(* IEC 61131-3 sources: ironplc-benchmarks/compat_out (part 59) *)

returs the date of january 1st for the given year
the function works for dates from 1970 - 2099

*)
(* @END_DECLARATION := '0' *)
YEAR_BEGIN := DWORD_TO_DATE(SHR(INT_TO_DWORD(y) * 1461 - 2878169,2) * 86400);

(* revision history
hm	19. dec 2007	rev 1.0
	original version

hm	4. jan 2008		rev 1.1
	formula for step7 was incorrect during leap years

hm	7. apr. 2008	rev 1.2
	deleted unused step7 code
*)

END_FUNCTION

(* @NESTEDCOMMENTS := 'Yes' *)
(* @PATH := '\/Time&Date' *)
(* @OBJECTFLAGS := '0, 8' *)
(* @SYMFILEFLAGS := '2048' *)
FUNCTION YEAR_END : DATE
VAR_INPUT
	y : INT;
END_VAR

(*
version 1.1	24. jan. 2011
programmer 	hugo
tested by	oscat

returs the date of december 31st for the given year
the function works for dates from 1970 - 2099

*)
(* @END_DECLARATION := '0' *)
YEAR_END := DWORD_TO_DATE(SHR(INT_TO_DWORD(y) * 1461 - 2876712, 2) * 86400);

(* revision history
hm	15. jun. 2008	rev 1.0
	original version

hm	24. jan 2011	rev 1.1
	improved performance
*)

END_FUNCTION

(* @NESTEDCOMMENTS := 'Yes' *)
(* @PATH := '\/Time&Date' *)
(* @OBJECTFLAGS := '0, 8' *)
(* @SYMFILEFLAGS := '2048' *)
FUNCTION YEAR_OF_DATE : INT
VAR_INPUT
	IDATE : DATE;
END_VAR

(*
version 1.4	7. oct. 2008
programmer 	hugo
tested by		oscat

returs the year of a date
the function works for dates from 1970 - 2099

*)

(* @END_DECLARATION := '0' *)
YEAR_OF_DATE := DWORD_TO_INT((DATE_TO_DWORD(idate) + 43200) / 31557600 + 1970);

(* revision history
hm	4. aug 2006		rev 1.0
	original version

hm	1. okt 2007		rev 1.1
	corrected error in algorithm
	adjustment for S7 compatibility

hm	23.12.2007		rev 1.2
	changed code for better performance

hm	7. apr. 2008	rev 1.3
	deleted unused step7 code

hm	7. oct. 2008	rev 1.4
	renamed function (year) to year_of_date

*)
END_FUNCTION

(* @NESTEDCOMMENTS := 'Yes' *)
(* @PATH := '' *)
(* @OBJECTFLAGS := '0, 8' *)
TYPE CALENDAR :
STRUCT
	UTC : DT;					(* world time UTC *)
	LDT : DT;					(* local time *)
	LDATE : DATE;				(* local date *)
	LTOD : TOD;					(* local time of day *)
	YEAR : INT;					(* year of LDATE *)
	MONTH : INT;				(* month of LDATE *)
	DAY : INT;					(* day of LDATE *)
	WEEKDAY : INT;				(* weekday of LDATE *)
	OFFSET : INT;				(* Time Zone Offset for Local time in minutes *)
	DST_EN : BOOL;				(* daylight savings time enable *)
	DST_ON : BOOL;				(* true when daylight savings time os on *)
	NAME : STRING[5];			(* name of time zone *)
	LANGUAGE : INT;			(* location number pls see location setup *)
	LONGITUDE : REAL;			(* longitude of current location *)
	LATITUDE : REAL;			(* latitude of current location *)
	SUN_RISE : TOD;				(* sun_rise for current location *)
	SUN_SET : TOD;				(* sun_set for current location *)
	SUN_MIDDAY : TOD;			(* worldtime when sun stands at south position *)
	SUN_HEIGTH : REAL	;		(* suns heigth at midday, south position *)
	SUN_HOR : REAL;			(* sun angle horizontal 0 = north in degrees *)
	SUN_VER : REAL;			(* sun angle vertical above horizon in degrees *)
	NIGHT : BOOL;				(* true between sun_set and sun_rise *)
	HOLIDAY : BOOL;			(* true when holiday *)
	HOLY_NAME : STRING[30];	(* name of holiday *)
	WORK_WEEK : INT;			(* current work week *)
END_STRUCT
END_TYPE

(* revision history
hm	21. nov. 2008	rev 1.0
	original version

hm	8. feb. 2009	rev 1.1
	added sun position data

hm	10. mar. 2009	rev 1.2
	added work_week, sun_midday, sun_heigth

hm	23. jan 2010	rev 1.3
	sun_rise, sun_set and sun_midday are now calculated in local time

*)
(* @END_DECLARATION := '0' *)

(* @NESTEDCOMMENTS := 'Yes' *)
(* @PATH := '' *)
(* @OBJECTFLAGS := '0, 8' *)
TYPE COMPLEX :
STRUCT
	re : REAL;
	im : REAL;
END_STRUCT
END_TYPE

(* revision history
hm	18. oct. 2008
	original version

*)
(* @END_DECLARATION := '0' *)

(* @NESTEDCOMMENTS := 'Yes' *)
(* @PATH := '' *)
(* @OBJECTFLAGS := '0, 8' *)
TYPE CONSTANTS_LANGUAGE :
STRUCT
	(* Language Setup *)
	DEFAULT : INT := 1; (* 1=english, 2=german 3=french *)
	LMAX : INT := 3;
	WEEKDAYS : ARRAY[1..3, 1..7] OF STRING[10] :=	['Monday', 'Tuesday', 'Wednesday', 'Thursday', 'Friday', 'Saturday', 'Sunday',
													'Montag', 'Dienstag', 'Mittwoch', 'Donnerstag', 'Freitag', 'Samstag', 'Sonntag',
													'Lundi', 'Mardi', 'Mercredi', 'Jeudi', 'Vendredi', 'Samedi', 'Dimanche'];
	WEEKDAYS2 : ARRAY[1..3, 1..7] OF STRING[2] :=	['Mo', 'Tu', 'We', 'Th', 'Fr', 'Sa', 'Su',
													'Mo', 'Di', 'Mi', 'Do', 'Fr', 'Sa', 'So',
													'Lu', 'Ma', 'Me', 'Je', 'Ve', 'Sa', 'Di'];
	MONTHS : ARRAY[1..3, 1..12] OF STRING[10] :=	['January', 'February', 'March', 'April', 'May', 'June', 'July', 'August', 'September', 'October', 'November', 'December',
													'Januar', 'Februar', 'M�rz', 'April', 'Mai', 'Juni', 'Juli', 'August', 'September', 'Oktober', 'November', 'Dezember',
													'Janvier', 'F�vrier', 'mars', 'Avril', 'Mai', 'Juin', 'Juillet', 'Ao�t', 'Septembre', 'Octobre', 'Novembre', 'Decembre'];
	MONTHS3 : ARRAY[1..3, 1..12] OF STRING[3] :=	['Jan', 'Feb', 'Mar', 'Apr', 'May', 'Jun', 'Jul', 'Aug', 'Sep', 'Oct', 'Nov', 'Dec',
													'Jan', 'Feb', 'Mrz', 'Apr', 'Mai', 'Jun', 'Jul', 'Aug', 'Sep', 'Okt', 'Nov', 'Dez',
													'Jan', 'Fev', 'Mar', 'Avr', 'Mai', 'Jun', 'Jul', 'Aou', 'Sep', 'Oct', 'Nov', 'Dec'];
	DIRS : ARRAY[1..3,0..15] OF STRING[3] :=		['N', 'NNE', 'NE', 'ENE', 'E', 'ESE', 'SE', 'SSE', 'S', 'SSW', 'SW', 'WSW', 'W', 'WNW', 'NW', 'NNW',
													'N', 'NNO', 'NO', 'ONO', 'O', 'OSO', 'SO', 'SSO', 'S', 'SSW', 'SW', 'WSW', 'W', 'WNW', 'NW', 'NNW',
													'N', 'NNO', 'NO', 'ONO', 'O', 'OSO', 'SO', 'SSO', 'S', 'SSW', 'SW', 'WSW', 'W', 'WNW', 'NW', 'NNW'];
END_STRUCT
END_TYPE

(* revision history
hm	19. oct. 2008	rev 1.0
	original version

hm	22. oct. 2008	rev 1.1
	added directions DIRS

hm	23. dec. 2008	rev 1.2
	added french language

*)
(* @END_DECLARATION := '0' *)

(* @NESTEDCOMMENTS := 'Yes' *)
(* @PATH := '' *)
(* @OBJECTFLAGS := '0, 8' *)
TYPE CONSTANTS_LOCATION :
STRUCT
	(* location setup *)
	DEFAULT : INT := 1; (* 1=germany, 2=austria 3=france 4=belgium-german 5= italien-S�dtirol *)
	LMAX : INT := 5;

	(* language spoken in the location *)
	LANGUAGE : ARRAY[1..5] OF INT := [2, 2, 3, 2, 2];

END_STRUCT
END_TYPE

(* revision history
hm	20. oct. 2008	rev 1.0
	original version

hm	23. dec. 2008	rev 1.1
	added french holidays

hm	18. jan 2011	rev 1.2
	added spoken language
	deleted holidays from structure for more flexibility

*)
(* @END_DECLARATION := '0' *)

(* @NESTEDCOMMENTS := 'Yes' *)
(* @PATH := '' *)
(* @OBJECTFLAGS := '0, 8' *)
TYPE CONSTANTS_MATH :
STRUCT
	PI : REAL := 	3.14159265358979323846264338327950288;		(* Kreiszahl PI *)
	PI2 : REAL := 	6.28318530717958647692528676655900576;	(* PI * 2 *)
	PI4 : REAL :=  12.56637061435917295385057353311801152;	(* PI * 4 *)
	PI05 : REAL :=  1.5707963267949;							(* PI / 2 *)
	PI025 : REAL := 0.785398163397448;							(* PI / 4 *)
	PI_INV : REAL := 0.318309886183791;						(* 1 / PI *)
	E : REAL := 	2.71828182845904523536028747135266249;		(* Euler constant e *)
	E_INV : REAL := 0.367879441171442;							(* 1 / e *)
	SQ2 : REAL :=	1.4142135623731;							(* Wurzel von 2 *)
	FACTS : ARRAY[0..12] OF DINT := [1,1,2,6,24,120,720,5040,40320,362880,3628800,39916800,479001600];
END_STRUCT
END_TYPE

(* revision history
hm	26.10.2008	rev 1.0
	original version

hm	26. mar. 2011	rev 1.1
	added array facts
*)
(* @END_DECLARATION := '0' *)

(* @NESTEDCOMMENTS := 'Yes' *)
(* @PATH := '' *)
(* @OBJECTFLAGS := '0, 8' *)
TYPE CONSTANTS_PHYS :
STRUCT
	C : REAL := 299792458.0;				(* Lichtgeschwindigkeit in m/s *)
	E : REAL := 1.60217653E-19;				(* elementarladung in Colomb = A * s *)
	G : REAL := 9.80665; 						(* Erdbeschleunigung in m / s� *)
	T0 : REAL := -273.15;						(* absoluter Nullpunkt in �C *)
	RU : REAL := 8.314472; 					(* Universelle Gaskonstante in J / (mol � K) *)
	PN : REAL := 101325.0;					(* NormalDruck in Pa *)
END_STRUCT
END_TYPE

(* revision history
hm	18.10.2008	rev 1.0
	original version

hm	13. mar. 2009	rev 1.1
	real constants updated to new systax using dot

*)
(* @END_DECLARATION := '0' *)

(* @NESTEDCOMMENTS := 'Yes' *)
(* @PATH := '' *)
(* @OBJECTFLAGS := '0, 8' *)
TYPE CONSTANTS_SETUP :
STRUCT
	(* setup Parameters *)
	EXTENDED_ASCII : BOOL := TRUE;
	CHARNAMES : ARRAY[1..4] OF STRING[253] := [';"&quot;&&amp;<&lt;>&gt;�&euro;�&nbsp;�&iexcl;�&cent;�&pound;�&curren;�&yen;�&brvbar;�&sect;�&uml;�&copy;�&ordf;�&laquo;�&not;�&shy;�&reg;�&macr;�&deg;�&plusmn;�&sup2;�&sup3;�&acute;�&micro;�&para;�&middot;�&cedil;�&sup1;�&ordm;�&raquo;�&frac14;�&Ucirc;',
		';�&frac34;�&iquest;�&Agrave;�&Aacute;�&Acirc;�&Atilde;�&Auml;�&Aring;�&AElig;�&Ccedil;�&Egrave;�&Eacute;�&Ecirc;�&Euml;�&Igrave;�&Iacute;�&Icirc;�&Iuml;�&ETH;�&Ntilde;�&Ograve;�&Oacute;�&Ocirc;�&Otilde;�&Ouml;�&times;�&Oslash;�&Ugrave;�&Uacute;�&frac12;',
		';�&Uuml;�&Yacute;�&THORN;�&szlig;�&agrave;�&aacute;�&acirc;�&atilde;�&auml;�&aring;�&aelig;�&ccedil;�&egrave;�&eacute;�&ecirc;�&euml;�&igrave;�&iacute;�&icirc;�&iuml;�&eth;�&ntilde;�&ograve;�&oacute;�&ocirc;�&otilde;�&ouml;�&divide;�&oslash;�&ugrave;',
		';�&uacute;�&ucirc;�&uuml;�&yacute;�&thorn;�&yuml;'];
	MTH_OFS : ARRAY[1..12] OF INT := [0,31,59,90,120,151,181,212,243,273,304,334];
	DECADES : ARRAY[0..8] OF REAL := [1.0,10.0,100.0,1000.0,10000.0,10000.0,100000.0,1000000.0,10000000.0];
END_STRUCT
END_TYPE

(* revision history
hm	24.10.2008	rev 1.0
	original version

*)
(* @END_DECLARATION := '0' *)

(* @NESTEDCOMMENTS := 'Yes' *)
(* @PATH := '' *)
(* @OBJECTFLAGS := '0, 8' *)
TYPE ESR_DATA :
STRUCT
	TYP : BYTE;
	ADRESS : STRING[10];
	DS : DT;
	TS : TIME;
	DATA : ARRAY[0..7] OF BYTE;
END_STRUCT
END_TYPE

(* revision history
hm	18. oct. 2008
	original version

*)
(* @END_DECLARATION := '0' *)

(* @NESTEDCOMMENTS := 'Yes' *)
(* @PATH := '' *)
(* @OBJECTFLAGS := '0, 8' *)
TYPE FRACTION :
STRUCT
	NUMERATOR : INT;
	DENOMINATOR : INT;
END_STRUCT
END_TYPE
(* @END_DECLARATION := '0' *)

(* @NESTEDCOMMENTS := 'Yes' *)
(* @PATH := '' *)
(* @OBJECTFLAGS := '0, 8' *)
TYPE HOLIDAY_DATA :
STRUCT
	NAME : STRING[30];
	DAY : SINT;
	MONTH : SINT;
	USE : SINT;
END_STRUCT
END_TYPE

(* revision history
hm	18. oct. 2008
	original version

*)

(*	if month = 0 then F_day is the offset in days from easter
	used :0 = NOT used, 1 = used, -1..-7 menas the weekday before the specified DATE example -3 means wednesday before 23.11
*)

(* samples for Holiday data

	HOLIDAY_DE : ARRAY[0..29] OF HOLIDAY_DATA := (name := 'Neujahr', day := 1, month := 1, use := 1),
		(name := 'Heilig Drei K�nige', day := 6, month := 1, use := 1),
		(name := 'Karfreitag', day := -2, month := 0, use := 1),
		(name := 'Ostersonntag', day := 0, month := 0, use := 1),
		(name := 'Ostermontag', day := 1, month := 0, use := 1),
		(name := 'Tag der Arbeit', day := 1, month := 5, use := 1),
		(name := 'Christi Himmelfahrt', day := 39, month := 0, use := 1),
		(name := 'Pfingstsonntag', day := 49, month := 0, use := 1),
		(name := 'Pfingstmontag', day := 50, month := 0, use := 1),
		(name := 'Fronleichnam', day := 60, month := 0, use := 1),
		(name := 'Augsburger Friedensfest', day := 8, month := 8, use := 0),
		(name := 'Maria Himmelfahrt', day := 15, month := 8, use := 1),
		(name := 'Tag der Deutschen Einheit', day := 3, month := 10, use := 1),
		(name := 'Reformationstag', day := 31, month := 10, use := 0),
		(name := 'Allerheiligen', day := 1, month := 11, use := 1),
		(name := 'Buss und Bettag', day := 23, month := 11, use := 0),
		(name := '1. Weihnachtstag', day := 25, month := 12, use := 1),
		(name := '2. Weihnachtstag', day := 26, month := 12, use := 1);

	HOLIDAY_AT : ARRAY[0..29] OF HOLIDAY_DATA := (name := 'Neujahr', day := 1, month := 1, use := 1),
		(name := 'Heilig Drei K�nige', day := 6, month := 1, use := 1),
		(name := 'Karfreitag', day := -2, month := 0, use := 1),
		(name := 'Ostersonntag', day := 0, month := 0, use := 1),
		(name := 'Ostermontag', day := 1, month := 0, use := 1),
		(name := '', day := 1, month := 5, use := 0),
		(name := 'Christi Himmelfahrt', day := 39, month := 0, use := 1),
		(name := 'Pfingstsonntag', day := 49, month := 0, use := 1),
		(name := 'Pfingstmontag', day := 50, month := 0, use := 1),
		(name := 'Fronleichnam', day := 60, month := 0, use := 1),
		(name := '', day := 8, month := 8, use := 0),
		(name := 'Maria Himmelfahrt', day := 15, month := 8, use := 1),
		(name := '', day := 3, month := 10, use := 0),
		(name := '', day := 31, month := 10, use := 0),
		(name := 'Allerheiligen', day := 1, month := 11, use := 1),
		(name := 'Maria Empf�ngnis', day := 8, month := 12, use := 1),
		(name := '1. Weihnachtstag', day := 25, month := 12, use := 1),
		(name := '2. Weihnachtstag', day := 26, month := 12, use := 1);

	HOLIDAY_FR : ARRAY[0..29] OF HOLIDAY_DATA := (name := 'Nouvel an', day := 1, month := 1, use := 1),
		(name := 'St Valentin', day := 14, month := 2, use := 0),
		(name := 'Vendredi Saint (alsace)', day := -2, month := 0, use := 0),
		(name := 'Dimanche de p�ques', day := 0, month := 0, use := 1),
		(name := 'Lundi de p�ques', day := 1, month := 0, use := 1),
		(name := 'Jeudi de Ascension', day := 39, month := 0, use := 1),
		(name := 'dimanche de Pentec�te ', day := 49, month := 0, use := 1),
		(name := 'jeudi de la Trinit�', day := 60, month := 0, use := 0),
		(name := 'F�te du travail', day := 1, month := 5, use := 1),
		(name := 'Victoire 1945 ', day := 8, month := 5, use := 1),
		(name := 'Prise de La bastille', day := 14, month := 7, use := 1),
		(name := '15 Ao�t 1944', day := 15, month := 8, use := 1),
		(name := 'Halloween', day := 31, month := 10, use := 0),
		(name := 'Armistice 1918', day := 11, month := 11, use := 1),
		(name := 'No�l', day := 25, month := 12, use := 1),
		(name := 'Saint �tienne (alsace)', day := 26, month := 12, use := 0),
		(name := 'F�te de la musique', day := 21, month := 6, use := 0);

	HOLIDAY_BED : ARRAY[0..29] OF HOLIDAY_DATA :=	(name := 'Neujahr', day := 1, month := 1, use := 1),
		(name := 'Ostersonntag', day := 0, month := 0, use := 1),
		(name := 'Ostermontag', day := 1, month := 0, use := 1),
		(name := 'Tag der Arbeit', day := 1, month := 5, use := 1),
		(name := 'Christi Himmelfahrt', day := 39, month := 0, use := 1),
		(name := 'Pfingsten', day := 49, month := 0, use := 1),
		(name := 'Pfingstmontag', day := 50, month := 0, use := 1),
		(name := 'Nationalfeiertag', day := 21, month := 7, use := 1),
		(name := 'Mari� Himmelfahrt', day := 15, month := 8, use := 1),
		(name := 'Allerheiligen', day := 1, month := 11, use := 1),
		(name := 'Feiertag DG', day := 15, month := 11, use := 1),
		(name := 'Heiligabend', day := 24, month := 12, use := 1),
		(name := '1. Weihnachtstag', day := 25, month := 12, use := 1),
		(name := '2. Weihnachtstag', day := 26, month := 12, use := 1),
		(name := 'Silvester', day := 31, month := 12, use := 1);

	HOLIDAY_ITD : ARRAY[0..29] OF HOLIDAY_DATA := (name := 'Neujahr', day := 1, month := 1, use := 1),
		(name := 'Heilig Drei K�nige', day := 6, month := 1, use := 1),
		(name := 'Ostersonntag', day := 0, month := 0, use := 1),
		(name := 'Ostermontag', day := 1, month := 0, use := 1),
		(name := 'Tag der Befeiung Italiens', day := 25, month := 4, use := 1),
		(name := 'Tag der Arbeit', day := 1, month := 5, use := 1),
		(name := 'Pfingsten', day := 49, month := 0, use := 1),
		(name := 'Pfingstmontag', day := 50, month := 0, use := 1),
		(name := 'Tag der Republik Italien', day := 2, month := 6, use := 1),
		(name := 'Mari� Himmelfahrt', day := 15, month := 8, use := 1),
		(name := 'Allerheiligen', day := 1, month := 11, use := 1),
		(name := 'Mari� Empf�ngnis', day := 8, month := 12, use := 1),
		(name := 'Heiligabend', day := 24, month := 12, use := 0),
		(name := '1. Weihnachtstag', day := 25, month := 12, use := 1),
		(name := '2. Stephanstag', day := 26, month := 12, use := 1);

*)
(* @END_DECLARATION := '0' *)

(* @NESTEDCOMMENTS := 'Yes' *)
(* @PATH := '' *)
(* @OBJECTFLAGS := '0, 8' *)
TYPE REAL2 :
STRUCT
	R1 : REAL;	(* small value *)
	RX : REAL;	(* big value *)
END_STRUCT
END_TYPE

(* revision history
hm	18. oct. 2008
	original version

*)
(* @END_DECLARATION := '0' *)

(* @NESTEDCOMMENTS := 'Yes' *)
(* @PATH := '' *)
(* @OBJECTFLAGS := '0, 8' *)
TYPE SDT :
STRUCT
	YEAR : INT;
	MONTH : INT;
	DAY : INT;
	WEEKDAY : INT;
	HOUR : INT;
	MINUTE : INT;
	SECOND : INT;
	MS : INT;
END_STRUCT
END_TYPE

(* revision history
hm	18. oct. 2008
	original version

*)
(* @END_DECLARATION := '0' *)

(* @NESTEDCOMMENTS := 'Yes' *)
(* @PATH := '' *)
(* @OBJECTFLAGS := '0, 8' *)
TYPE TIMER_EVENT :
STRUCT
	TYP : BYTE;
	CHANNEL : BYTE;
	DAY : BYTE;
	START : TOD;
	DURATION : TIME;
	LAND : BYTE;
	LOR : BYTE;
	LAST : DT;
END_STRUCT
END_TYPE

(* revision history
hm	18. oct. 2008	rev 1.0
	original version

hm	26. jan. 2011	rev 1.1
	changed type of last to be DT
*)
(* @END_DECLARATION := '0' *)

(* @NESTEDCOMMENTS := 'Yes' *)
(* @PATH := '' *)
(* @OBJECTFLAGS := '0, 8' *)
TYPE VECTOR_3 :
STRUCT
	X : REAL;
	Y : REAL;
	Z : REAL;
END_STRUCT
END_TYPE

(* revision history
hm	18. oct. 2008
	original version

*)
(* @END_DECLARATION := '0' *)

(* @NESTEDCOMMENTS := 'Yes' *)
(* @GLOBAL_VARIABLE_LIST := 'Constants' *)
(* @PATH := '' *)
(* @OBJECTFLAGS := '0, 8' *)
(* @SYMFILEFLAGS := '4096' *)
VAR_GLOBAL CONSTANT
	STRING_LENGTH : INT := 250;
	LIST_LENGTH : INT := 250;
END_VAR

(* revisionhistory
hm 3. mar. 2007
	extended accuracy of pi2
	renamed T0 to Tk for better compatibility with other libraries
	renamed C t0 c0 for better compatibility

hm	2. may. 2007
	added RU universal gas constant

hm	1. oct. 2007
	added setup parameter STEP7

hm 31. oct. 2007
	added PN

hm	6. mar. 2008
	added setup Parameter EXTENDED_ASCII

hm	28. Mar. 2008
	added setup parameter STRING_LENGTH

hm	7. apr. 2008
	Deleted unused setup parameter Step7

hm	19. apr. 2008
	added setup parameter NETWORK_BUFFER_SIZE

hm	27. apr. 2008
	added PI05 and PI025

hm	18. may. 2008
	added charname lists
	renamed E to E1

hm	30. jun. 2008
	reduced size of string constants to 253 to avoid problems with target aixia DCUF

hm	21. sep. 2008
	added section language setup
	added section location setup

hm	20. oct. 2008
	changed to structured constants

hm	16. nov. 2008
	moved structured constants to global vars for compatibility reasons

hm	13. nov. 2009
	added network_buffer_short_size
	renamed network_buffer_long_size
	changed string length to 250

hm	20. jan. 2011
	removed network buffers
	added list_length
*)
(* @OBJECT_END := 'Constants' *)
(* @CONNECTIONS := Constants
FILENAME : ''
FILETIME : 0
EXPORT : 0
NUMOFCONNECTIONS : 0
*)

(* @NESTEDCOMMENTS := 'Yes' *)
(* @GLOBAL_VARIABLE_LIST := 'Globale_Variablen' *)
(* @PATH := '' *)
(* @OBJECTFLAGS := '0, 8' *)
(* @SYMFILEFLAGS := '4096' *)
VAR_GLOBAL
	MATH : CONSTANTS_MATH;
	PHYS : CONSTANTS_PHYS;
	LANGUAGE : CONSTANTS_LANGUAGE;
	SETUP : CONSTANTS_SETUP;
	LOCATION : CONSTANTS_LOCATION;
END_VAR
(* @OBJECT_END := 'Globale_Variablen' *)
(* @CONNECTIONS := Globale_Variablen
FILENAME : ''
FILETIME : 0
EXPORT : 0
NUMOFCONNECTIONS : 0
*)

(* @NESTEDCOMMENTS := 'Yes' *)
(* @GLOBAL_VARIABLE_LIST := 'Setup_Data' *)
(* @PATH := '' *)
(* @OBJECTFLAGS := '0, 8' *)
(* @SYMFILEFLAGS := '4096' *)
VAR_GLOBAL RETAIN

END_VAR

(* @OBJECT_END := 'Setup_Data' *)
(* @CONNECTIONS := Setup_Data
FILENAME : ''
FILETIME : 0
EXPORT : 0
NUMOFCONNECTIONS : 0
*)

/* LIBRARY */
/* Standard.lib 4.10.05 11:14:46 */
/* (* @LIBRARYSYMFILEINFO := '0' *) */
/* NumOfPOUs: 21 */
/* CONCAT: 0 */
/* CTD: 0 */
/* CTU: 0 */
/* CTUD: 0 */
/* DELETE: 0 */
/* F_TRIG: 0 */
/* FIND: 0 */
/* INSERT: 0 */
/* LEFT: 0 */
/* LEN: 0 */
/* MID: 0 */
/* R_TRIG: 0 */
/* REPLACE: 0 */
/* RIGHT: 0 */
/* RS: 0 */
/* RTC: 0 */
/* SEMA: 0 */
/* SR: 0 */
/* TOF: 0 */
/* TON: 0 */
/* TP: 0 */
/* NumOfGVLs: 0 */
/* END_LIBRARY */

PROGRAM test_BAND_B
VAR
    result : BYTE;
END_VAR
    result := BAND_B(X := BYTE#16#AA, B := BYTE#16#AA);
END_PROGRAM

(* ---- test_BCDC_TO_INT.st ---- *)
(* IronPLC Compatibility Library

   Provides CODESYS-specific functions that are not part of IEC 61131-3
   and not built into IronPLC, but are needed by the OSCAT library.

   These are prepended to the compilation unit when running the
   compatibility test with --lib.
*)

(* Byte_of_Dword: Extract a byte from a DWORD by index.
   N=0 is the least significant byte, N=3 is the most significant.
   CODESYS built-in, used 16 times in OSCAT. *)
FUNCTION Byte_of_Dword : BYTE
VAR_INPUT
    in : DWORD;
    N : BYTE;
END_VAR
    Byte_of_Dword := DWORD_TO_BYTE(SHR(in, BYTE_TO_INT(N) * 8));
END_FUNCTION

(* DAY_OF_WEEK: Return day of week for a DATE value.
   Returns 0=Sunday, 1=Monday, ..., 6=Saturday.
   CODESYS extension, used 12 times in OSCAT.
   DATE is seconds since 1970-01-01. Jan 1 1970 was Thursday (=4). *)
FUNCTION DAY_OF_WEEK : SINT
VAR_INPUT
    in : DATE;
END_VAR
VAR
    days : DINT;
END_VAR
    days := DWORD_TO_DINT(DATE_TO_DWORD(in) / 86400);
    DAY_OF_WEEK := DINT_TO_SINT(((days MOD 7) + 4) MOD 7);
END_FUNCTION

(* TIME: Return current PLC uptime.
   CODESYS built-in, used 2 times in OSCAT.
   NOTE: Returns T#0s stub because __SYSTEM_UP_TIME is not accessible
   from FUNCTION context. Runtime value will not be correct until
   global variable access from functions is supported. *)
FUNCTION TIME : TIME
    TIME := T#0s;
END_FUNCTION

(* @NESTEDCOMMENTS := 'Yes' *)
(* @PATH := '\/Buffer Management' *)
(* @OBJECTFLAGS := '0, 8' *)
(* @SYMFILEFLAGS := '2048' *)
FUNCTION _BUFFER_CLEAR : BOOL
VAR_INPUT
	PT : REF_TO BYTE;
	SIZE : UINT;
END_VAR
VAR
	ptw : REF_TO DWORD;
	temp: LWORD;
	end, end32 : DWORD;
END_VAR

(*
version 1.2	31. oct. 2008
programmer 	hugo
tested by	oscat

this function will initialize a given array of byte with 0.
the function needs to be called:	_buffer_clear(adr("array"),sizeof("array"));
this function will manipulate a given array.
the function manipulates the original array, it rerturnes true when finished.
because this function works with pointers its very time efficient and it needs no extra memory.

*)
(* @END_DECLARATION := '0' *)
(* this routine uses 32 bit access to gain speed *)
(* first access bytes till pointer is aligned for 32 bit access *)
temp := pt;
end := temp + UINT_TO_DWORD(size);
end32 := end - 3;
WHILE (pt < end) AND ((temp AND 16#00000003) > 0) DO
	pt^ := 0;
	pt := pt + 1;
	temp := temp + 1;
END_WHILE;
(* pointer is aligned, now copy 32 bits at a time *)
ptw := pt;
WHILE ptw < end32 DO (* *)
	ptw^ := 0;
	ptw := ptw + 4;
END_WHILE;
(* copy the remaining bytes in byte mode *)
pt := ptw;
WHILE pt < end DO
	pt^ := 0;
	pt := pt + 1;
END_WHILE;

_BUFFER_CLEAR := TRUE;

(* revision History
hm 	5. mar. 2008	rev 1.0
	original version

hm	16. mar. 2008	rev 1.1
	added type conversion to avoid warnings under codesys 30
	chaged type of input size to uint
	deleted unused variable i

hm	31. oct. 2008	rev 1.2
	corrected an error while routine would write outside of arrays

*)
END_FUNCTION

(* @NESTEDCOMMENTS := 'Yes' *)
(* @PATH := '\/Buffer Management' *)
(* @OBJECTFLAGS := '0, 8' *)
(* @SYMFILEFLAGS := '2048' *)
FUNCTION _BUFFER_INIT : BOOL
VAR_INPUT
	PT : REF_TO BYTE;
	SIZE : UINT;
	INIT : BYTE;
END_VAR
VAR
	ptw : REF_TO DWORD;
	temp : LWORD;
	end, end32 : DWORD;
END_VAR

(*
version 1.2	31. oct. 2008
programmer 	hugo
tested by	oscat

this function will initialize a given array of byte with init.
the function needs to be called:	_buffer_init(adr("array"),sizeof("array"),init);
this function will manipulate a given array.
the function manipulates the original array, it rerturnes true when finished.
because this function works with pointers its very time efficient and it needs no extra memory.

*)
(* @END_DECLARATION := '0' *)
(* this routine uses 32 bit access to gain speed *)
(* first access bytes till pointer is aligned for 32 bit access *)
temp := pt;
end := temp + UINT_TO_DWORD(size);
end32 := end - 3;
WHILE (pt < end) AND ((temp AND 16#00000003) > 0) DO
	pt^ := init;
	pt := pt + 1;
	temp := temp + 1;
END_WHILE;
(* pointer is aligned, now copy 32 bits at a time *)
ptw := pt;
temp := SHL(BYTE_TO_DWORD(init),24) OR SHL(BYTE_TO_DWORD(init),16) OR SHL(BYTE_TO_DWORD(init),8) OR BYTE_TO_DWORD(init);
WHILE ptw < end32 DO
	ptw^ := temp;
	ptw := ptw + 4;
END_WHILE;
(* copy the remaining bytes in byte mode *)
pt := ptw;
WHILE pt < end DO
	pt^ := init;
	pt := pt + 1;
END_WHILE;

_BUFFER_INIT := TRUE;

(* revision History
hm 	5. mar. 2008	rev 1.0
	original version

hm	16. mar. 2008	rev 1.1
	added type conversion to avoid warnings under codesys 3.0
	chaged type of input size to uint.

hm	31. oct. 2008	rev 1.2
	corrected an error while routine would write outside of arrays

*)
END_FUNCTION

(* @NESTEDCOMMENTS := 'Yes' *)
(* @PATH := '\/Buffer Management' *)
(* @OBJECTFLAGS := '0, 8' *)
(* @SYMFILEFLAGS := '2048' *)
FUNCTION _BUFFER_INSERT : INT
VAR_INPUT
	STR : STRING[STRING_LENGTH];
	POS : INT;
	PT : REF_TO ARRAY[0..32767] OF BYTE;
	SIZE : UINT;
END_VAR
VAR
	end : INT;
	lx: INT;
	i: INT;
END_VAR

(*
version 1.5	2. jan. 2012
programmer 	hugo
tested by	oscat

this function will insert a string at a given position in a buffer.
the function needs to be called:	_buffer_init(adr("array"),sizeof("array"),init);
this function will manipulate a given array.
the function manipulates the original array, it returnes the next position after the input string when finished.
because this function works with pointers its very time efficient and it needs no extra memory.

*)
(* @END_DECLARATION := '0' *)
lx := LEN(str);
end := pos + lx;
(* first move the upper part of the buffer to make space for the string *)
FOR i := UINT_TO_INT(size) - 1 TO end BY -1 DO
	pt^[i] := pt^[i-lx];
END_FOR;
(* copy the string *)
_BUFFER_INSERT := _STRING_TO_BUFFER(str, pos, PT, size);

(* revision History
hm 	9. mar. 2008	rev 1.0
	original version

hm	16. mar. 2008	rev 1.1
	changed type of input size to uint

hm	13. may. 2008	rev 1.2
	changed type of pointer to array[1..32767]
	changed size of string to STRING_LENGTH

hm	23. mar. 2009	rev 1.3
	avoid writing to input pos

hm	12. nov. 2009	rev 1.4
	code optimized

hm 2. jan 2012	rev 1.5
	function now returns the next position after the input string

*)
END_FUNCTION

(* @NESTEDCOMMENTS := 'Yes' *)
(* @PATH := '\/Buffer Management' *)
(* @OBJECTFLAGS := '0, 8' *)
(* @SYMFILEFLAGS := '2048' *)
FUNCTION _BUFFER_UPPERCASE : BOOL
VAR_INPUT
	PT : REF_TO ARRAY[0..32000] OF BYTE;
	SIZE : INT;
END_VAR
VAR
	pos: INT;
END_VAR

(*
version 1.0	20. jan. 2011
programmer 	hugo
tested by	oscat

this function will convert an array of byte into uppercase
the function needs to be called:	_buffer_clear(adr("array"),sizeof("array"));
this function will manipulate a given array.
the function manipulates the original array, it rerturnes true when finished.
because this function works with pointers its very time efficient and it needs no extra memory.

*)
(* @END_DECLARATION := '0' *)
pos := 0;
WHILE pos < size DO
	PT^[pos] := TO_UPPER(pt^[pos]);
	pos := pos + 1;
END_WHILE;

_BUFFER_UPPERCASE := TRUE;

(* revision History
hm 	20. jan. 2011	rev 1.0
	original version

*)
END_FUNCTION

(* @NESTEDCOMMENTS := 'Yes' *)
(* @PATH := '\/Buffer Management' *)
(* @OBJECTFLAGS := '0, 8' *)
(* @SYMFILEFLAGS := '2048' *)
FUNCTION _STRING_TO_BUFFER : INT
VAR_INPUT
	STR : STRING[STRING_LENGTH];
	POS : INT;
	PT : REF_TO ARRAY[0..32767] OF BYTE;
	SIZE : UINT;
END_VAR
VAR
	ps : REF_TO BYTE;
	i: INT;
	end: INT;
END_VAR

(*
version 1.4	2. jan. 2012
programmer 	hugo
tested by		oscat

this function will copy a string into an array of byte starting at position pos.
the function needs to be called:	_String_To_buffer(str, pos, adr("array"),sizeof("array"));
this function will manipulate the array directly in memory and returns the position after the input string when finished.
because this function works with pointers its very time efficient and it needs no extra memory.

*)
(* @END_DECLARATION := '0' *)
ps := REF(str);
end := MIN(pos + LEN(str), UINT_TO_INT(size));
IF end > 0 THEN end := end -1; END_IF;
FOR i := pos TO end DO
	pt^[i] := ps^;
	ps := ps + 1;
END_FOR;

_STRING_TO_BUFFER := i;

(* revision History

hm 	5. mar. 2008	rev 1.0
	original version

hm	16. mar. 2008	rev 1.1
	changed type of input size to uint

hm	13. may. 2008	rev 1.2
	changed type of pointer to array[1..32767]
	changed size of string to STRING_LENGTH

hm	12. nov. 2009	rev 1.3
	limit end to size - 1

hm	2. jan 2012	rev 1.4
	return the position after the input string when finished
*)
END_FUNCTION

(* @NESTEDCOMMENTS := 'Yes' *)
(* @PATH := '\/Buffer Management' *)
(* @OBJECTFLAGS := '0, 8' *)
(* @SYMFILEFLAGS := '2048' *)
FUNCTION BUFFER_COMP : INT
VAR_INPUT
	PT1 : REF_TO ARRAY[0..32767] OF BYTE;
	SIZE1 : INT;
	PT2 : REF_TO ARRAY[0..32767] OF BYTE;
	SIZE2 : INT;
	START : INT;
END_VAR
VAR
	i, j, end : INT;
	firstbyte: BYTE;
END_VAR

(*
version 1.1	12. nov. 2009
programmer 	hugo
tested by	oscat

*)
(* @END_DECLARATION := '0' *)
(* search for first character match *)
IF size2 <= size1 THEN
	end := size1 - size2;
	firstbyte := PT2^[0];
	FOR i := START TO end DO
		IF PT1^[i] = firstbyte THEN
			(* first character matches, now compare rest of array *)
			j := 1;
			WHILE j < size2 DO
				IF pt2^[j] <> pt1^[j+i] THEN EXIT; END_IF;
				j := j + 1;
			END_WHILE;
			(* when J > size2 a match was found return the position i in buffer1 *)
			IF j = size2 THEN
				BUFFER_COMP := i;
				RETURN;
			END_IF;
		END_IF;
	END_FOR;
END_IF;
BUFFER_COMP := -1;

(*
hm 14. nov. 2008	rev 1.0
	original version

hm	12. nov. 2009	rev 1.1
	performance increase

*)
END_FUNCTION

(* @NESTEDCOMMENTS := 'Yes' *)
(* @PATH := '\/Buffer Management' *)
(* @OBJECTFLAGS := '0, 8' *)
(* @SYMFILEFLAGS := '2048' *)
FUNCTION BUFFER_SEARCH : INT
VAR_INPUT
	PT : REF_TO ARRAY[0..32767] OF BYTE;
	SIZE : INT;
	STR : STRING[STRING_LENGTH];
	POS : INT;
	IGN : BOOL;
END_VAR
VAR
	ps : REF_TO ARRAY[0..STRING_LENGTH] OF BYTE;
	chx : BYTE;
	i: INT;
	end: INT;
	k: INT;
	lx: INT;
END_VAR

(*
version 1.4	25. jan 2011
programmer 	hugo
tested by	oscat

this function will search for a string STR in an array of byte starting at position pos.
the function needs to be called: buffer_search(adr("array"),sizeof("array"), STR, POS, IGN);
because this function works with pointers its very time efficient and it needs no extra memory.
The function returns the position of the first character of the string in the array if found.
a -1 is returned if the string is not found in the array.
when IGN = TRUE, STR must be in capital letters and the search is case insensitv.

*)
(* @END_DECLARATION := '0' *)
ps := REF(STR);
lx := LEN(STR);
end := MIN(SIZE - lx, SIZE - 1);
lx := lx - 1;
FOR i := pos TO end DO
	FOR k := 0 TO lx DO
		IF IGN THEN chx := TO_UPPER(pt^[i+k]); ELSE chx := pt^[i+k]; END_IF;
		IF ps^[k] <> chx THEN EXIT; END_IF;
	END_FOR;
	IF k > lx THEN
		BUFFER_SEARCH := i;
		RETURN;
	END_IF;
END_FOR;
BUFFER_SEARCH := -1;

(* revision History

hm 5. mar. 2008	rev 1.0
	original version

hm	16. mar. 2008	rev 1.1
	chaged type of input size to uint

hm	13. may. 2008	rev 1.2
	changed type of pointer to array[1..32767]
	changed size of string to STRING_LENGTH

hm	12. nov. 2009	rev 1.3
	limit end to array size

hm	25. jan. 2011	rev 1.4
	ign = True will now ignore case
	return -1 if nothing found
*)
END_FUNCTION

(* @NESTEDCOMMENTS := 'Yes' *)
(* @PATH := '\/Buffer Management' *)
(* @OBJECTFLAGS := '0, 8' *)
(* @SYMFILEFLAGS := '2048' *)
FUNCTION BUFFER_TO_STRING : STRING[STRING_LENGTH]
VAR_INPUT
	PT : REF_TO ARRAY[0..32767] OF BYTE;
	SIZE : UINT;
	START : UINT;
	STOP : UINT;
END_VAR
VAR
	ps : REF_TO BYTE;
	i : UINT;
	stp: UINT;
	sta: UINT;
END_VAR

(*
version 1.5	12. nov. 2009
programmer 	hugo
tested by		oscat

this function will retrieve a string from an array of byte starting at position start and stop at position stop.
the function needs to be called:	buffer_TO_String(adr("array"),sizeof("array"), start, stop);
because this function works with pointers its very time efficient and it needs no extra memory.

*)
(* @END_DECLARATION := '0' *)
ps := REF(BUFFER_TO_STRING);
IF size = 0 THEN RETURN; END_IF;
sta := MIN(start, size -1);
stp := MIN(stop, size -1);

(* check for maximum string_length *)
IF UINT_TO_INT(stp - sta + 1) >= STRING_LENGTH THEN
	stp := sta + INT_TO_UINT(STRING_LENGTH) - 1;
END_IF;

FOR i := sta TO stp DO
	ps^ := pt^[i];
	ps := ps + 1;
END_FOR;

(* terminate the string *)

ps^ := 0;

(* revision History
hm 	5. mar. 2008	rev 1.0
	original version

hm	16. mar. 2008	rev 1.1
	changed type of input size to uint

hm	13. may. 2008	rev 1.2
	changed type of pointer to array[0..32767]
	changed size of string to STRING_LENGTH

hm	12. jun. 2008	rev 1.3
	check for pointer overrun
	change input start and stop to uint
	added type conversions to avoid warnings under codesys 3.0

hm	23. mar. 2009	rev 1.4
	avoid writing to input stop

hm	12. nov. 2009 rev 1.5
	limit start and stop to size -1

*)
END_FUNCTION

(* @NESTEDCOMMENTS := 'Yes' *)
(* @PATH := '\/Engineering\/automation' *)
(* @OBJECTFLAGS := '0, 8' *)
(* @SYMFILEFLAGS := '2048' *)
FUNCTION_BLOCK DRIVER_1
VAR_INPUT (* CONSTANT *)
	Toggle_Mode : BOOL;
	Timeout : TIME;
END_VAR
VAR_INPUT
	SET0 : BOOL;
	IN : BOOL;
	RST : BOOL;
END_VAR
VAR_OUTPUT
	Q : BOOL;
END_VAR
VAR
	off : TON;
	edge: BOOL;
END_VAR

(*
version 1.0	2 jan 2008
programmer 	hugo
tested by		tobias

driver_1 is a multi purpose driver.
a rising edge on in sets the output high if toggle is flase. while toggle is true, a rising edge on in toggles the output Q.
if a timeout is specified the output q will be reset to false automatically after the timeout has elapsed.
a asynchronous reset and set will force the output high or low respectively.

*)
(* @END_DECLARATION := '0' *)
IF off.Q THEN Q := FALSE; END_IF;
IF rst THEN
	Q := FALSE;
ELSIF set0 THEN
	Q := TRUE;
ELSIF IN AND NOT edge THEN
	IF toggle_mode THEN q := NOT Q; ELSE q := TRUE; END_IF;
END_IF;
edge := in;
IF timeout > t#0s THEN off(in := Q, PT := Timeout); END_IF;

(* revision history
hm	2. jan 2008		rev 1.0
	original version

*)
END_FUNCTION_BLOCK

(* @NESTEDCOMMENTS := 'Yes' *)
(* @PATH := '\/Engineering\/automation' *)
(* @OBJECTFLAGS := '0, 8' *)
(* @SYMFILEFLAGS := '2048' *)
FUNCTION_BLOCK DRIVER_4
VAR_INPUT (* CONSTANT *)
	Toggle_Mode : BOOL;
	Timeout : TIME;
END_VAR
VAR_INPUT
	SET0 : BOOL;
	IN0, IN1, IN2, IN3 : BOOL;
	RST : BOOL;
END_VAR
VAR_OUTPUT
	Q0, Q1, Q2, Q3 : BOOL;
END_VAR
VAR
	d0, d1, d2, d3 : DRIVER_1;
END_VAR

(*
version 1.0	2 jan 2008
programmer 	hugo
tested by		tobias

driver_4 is a 4 channel multi purpose driver.
a rising edge on in? sets the output Q? high if toggle_mode is flase. while toggle_mode is true, a rising edge on in? toggles the output Q?.
if a timeout is specified the output Q? will be reset to false automatically after the timeout has elapsed.
a asynchronous reset and set will force the output high or low respectively.
an asynchronous set will force all outputs high simultaneously

*)
(* @END_DECLARATION := '0' *)
D0(Set0:=set0, in:=in0, rst:=rst, toggle_mode:=toggle_mode, timeout:=timeout);
D1(Set0:=set0, in:=in1, rst:=rst, toggle_mode:=toggle_mode, timeout:=timeout);
D2(Set0:=set0, in:=in2, rst:=rst, toggle_mode:=toggle_mode, timeout:=timeout);
D3(Set0:=set0, in:=in3, rst:=rst, toggle_mode:=toggle_mode, timeout:=timeout);
Q0 := D0.Q;
Q1 := D1.Q;
Q2 := D2.Q;
Q3 := D3.Q;

(* revision history
hm	2. jan 2008		rev 1.0
	original version

*)
END_FUNCTION_BLOCK

(* @NESTEDCOMMENTS := 'Yes' *)
(* @PATH := '\/Engineering\/automation' *)
(* @OBJECTFLAGS := '0, 8' *)
(* @SYMFILEFLAGS := '2048' *)
FUNCTION_BLOCK DRIVER_4C
VAR_INPUT
	IN : BOOL;
	RST : BOOL;
END_VAR
VAR_INPUT (* CONSTANT *)
	Timeout : TIME;
	SX : ARRAY[1..7] OF BYTE := [1,3,7,15];
END_VAR
VAR_OUTPUT
	SN : INT;
	Q0 : BOOL;
	Q1 : BOOL;
	Q2 : BOOL;
	Q3 : BOOL;
END_VAR
VAR
	off : TON;
	edge: BOOL;
END_VAR

(*
version 1.0	23. mar. 2009
programmer 	hugo
tested by	tobias

driver_4C is a multi purpose driver.
a rising edge on in switches from S0 state S1 and the next edge to state S2 and so on.
in state S0 all outputs Q are FALSE.
The stet of the Outputs in any state S? is configurable with setup variables.
The variables S1..S5 define the states, while the sequence is terminated when a state Variable S? = 0.
The lower bits 0..3 of the state vars S? are corresponding to the Outputs Q0..Q3

*)
(* @END_DECLARATION := '0' *)
IF RST OR off.Q THEN
	SN := 0;
ELSIF IN AND NOT edge THEN
	SN := SN + 1;
	IF SN > 7 OR SX[SN] = 0 THEN SN := 0; END_IF;
END_IF;
edge := in;
IF SN > 0 THEN
	Q0 := SX[SN].0;
	Q1 := SX[SN].1;
	Q2 := SX[SN].2;
	Q3 := SX[SN].3;
ELSE
	Q0 := FALSE;
	Q1 := FALSE;
	Q2 := FALSE;
	Q3 := FALSE;
END_IF;

(* maximaum timeout *)
IF timeout > t#0s THEN off(in := SN > 0, PT := Timeout); END_IF;

(* revision history
hm	23. mar. 2009	rev 1.0
	original version

*)
END_FUNCTION_BLOCK

(* @NESTEDCOMMENTS := 'Yes' *)
(* @PATH := '\/Engineering\/automation' *)
(* @OBJECTFLAGS := '0, 8' *)
(* @SYMFILEFLAGS := '2048' *)
 FUNCTION_BLOCK FLOW_CONTROL
VAR_INPUT
	IN : BOOL;
	REQ : BOOL;
	ENQ : BOOL;
	RST : BOOL;
END_VAR
VAR_INPUT (* CONSTANT *)
	T_AUTO : TIME := T#1h;
	T_DELAY : TIME := T#23h;
END_VAR
VAR_OUTPUT
	Q : BOOL;
	STATUS : BYTE;
END_VAR
VAR
	timer : TP_1D;
END_VAR

(*
version 1.0	28. jun. 2008
programmer 	hugo
tested by	oscat

FLOW_CONTROL switches a valves depending on the input in.
flow control also limits the maximum ontime of the valve and controls pressure on the output side.

*)

(* @END_DECLARATION := '0' *)
STATUS := 100;
IF RST THEN
	Q := FALSE;
	timer(rst := TRUE);
	timer.RST := FALSE;
	STATUS := 103;
ELSIF ENQ THEN
	IF IN THEN
		status := 101;
	END_IF;
	IF REQ THEN
		(* timer will generate a timed pulse after TP goes high *)
		timer.PT1 := T_AUTO;
		timer.PTD := T_DELAY;
		timer.IN := TRUE;
		STATUS := 102;
	END_IF;
END_IF;

(* set output and run timer *)
timer();
timer.IN := FALSE;
Q := (IN AND ENQ) OR timer.Q;

(* revision history
hm 	28. jun. 2008 	rev 1.0
	original version

*)
END_FUNCTION_BLOCK

(* @NESTEDCOMMENTS := 'Yes' *)
(* @PATH := '\/Engineering\/automation' *)
(* @OBJECTFLAGS := '0, 8' *)
(* @SYMFILEFLAGS := '2048' *)
FUNCTION_BLOCK FT_Profile
VAR_INPUT
	K : REAL := 1.0;
	O : REAL;
	M : REAL := 1.0;
	E : BOOL;
END_VAR
VAR_INPUT (* CONSTANT *)
	value_0 : REAL;
	time_1 : TIME;
	value_1 : REAL;
	time_2 : TIME;
	value_2 : REAL;
	time_3 : TIME;
	value_3 : REAL;
	time_10 : TIME;
	value_10 : REAL;
	time_11 : TIME;
	value_11 : REAL;
	time_12 : TIME;
	value_12 : REAL;
	time_13 : TIME;
	value_13 : REAL;
END_VAR
VAR_OUTPUT
	Y : REAL;
	RUN : BOOL;
	ET : TIME;
END_VAR
VAR
	tx : TIME;
	edge : BOOL;
	state: BYTE;
	ta: TIME;
	tb: TIME;
	t0 : TIME;
	temp: REAL;
	va: REAL;
	vb: REAL;
END_VAR

(*
version 1.1	15 sep 2007
programmer 	tobias
tested by		hugo

FT_Profile generates an output signal which is defined by values over a time scale.
the different values are connected by ramps between the individual values.
a rising edge on E starts the output signal generation and E = True can delay time_3 / value_3 as long as it stays true.
an additional multiplier K can be used to multiply the output and an offset O can be added to the output dynamically.
*)
(* @END_DECLARATION := '0' *)
(* read system time *)
tx := DWORD_TO_TIME(T_PLC_MS());

(* determine start condition *)
IF E AND NOT edge THEN
	RUN := TRUE;
	ET := t#0s;
	t0 := tx;
	ta := tx;
	tb := multime(time_1, M);
	va := value_0;
	vb := value_1;
	temp := value_0;
	state := 1;
END_IF;
edge := E;

(* generate startup profile *)
IF run THEN
	CASE state OF
		1:	IF tx - ta >= tb THEN
				ta := ta + tb;
				tb := multime(time_2 - time_1, M);
				va := value_1;
				vb := value_2;
				temp := value_1;
				state := 2;
			ELSE
				temp := ((vb - va) * TIME_TO_REAL(tx - ta) / TIME_TO_REAL(tb) + va);
			END_IF;
		2:	IF tx - ta >= tb THEN
				ta := ta + tb;
				tb := multime(time_3 - time_2, M);
				va := value_2;
				vb := value_3;
				temp := value_2;
				state := 3;
			ELSE
				temp := ((vb - va) * TIME_TO_REAL(tx - ta) / TIME_TO_REAL(tb) + va);
			END_IF;
		3:	IF tx - ta >= tb THEN
				ta := ta + tb;
				tb := multime(time_10 - time_3, M);
				va := value_3;
				vb := value_10;
				temp := value_3;
				state := 4;
			ELSE
				temp := ((vb - va) * TIME_TO_REAL(tx - ta) / TIME_TO_REAL(tb) + va);
			END_IF;
		4 :	IF tx - ta >= tb THEN
				ta := ta + tb;
				tb := multime(time_11 - time_10, M);
				va := value_10;
				vb := value_11;
				temp := value_10;
				IF E THEN state := 5; ELSE state := 6; END_IF;
			ELSE
				temp := ((vb - va) * TIME_TO_REAL(tx - ta) / TIME_TO_REAL(tb) + va);
			END_IF;
		5:	(* extend the signal while E is true *)
			IF E THEN
				ta := tx;
			ELSE
				state := 6;
			END_IF;
		6:	IF tx - ta >= tb THEN
				ta := ta + tb;
				tb := multime(time_12 - time_11, M);
				va := value_11;
				vb := value_12;
				temp := value_11;
				state := 7;
			ELSE
				temp := ((vb - va) * TIME_TO_REAL(tx - ta) / TIME_TO_REAL(tb) + va);
			END_IF;
		7:	IF tx - ta >= tb THEN
				ta := ta + tb;
				tb := multime(time_13 - time_12, M);
				va := value_12;
				vb := value_13;
				temp := value_12;
				state := 8;
			ELSE
				temp := ((vb - va) * TIME_TO_REAL(tx - ta) / TIME_TO_REAL(tb) + va);
			END_IF;
		8:	IF tx - ta >= tb THEN
				temp := value_13;
				run := FALSE;
			ELSE
				temp := ((vb - va) * TIME_TO_REAL(tx - ta) / TIME_TO_REAL(tb) + va);
			END_IF;
	END_CASE;
	Y := temp * K + O;
	ET := tx - t0;
END_IF;

(* revision history
hm	27 feb 2007		rev 1.0
	original version

hm	15. sep2007		rev 1.1
	replaced Time() with T_PLC_MS for compatibility and performance reasons

*)
END_FUNCTION_BLOCK

(* @NESTEDCOMMENTS := 'Yes' *)
(* @PATH := '\/Engineering\/automation' *)
(* @OBJECTFLAGS := '0, 8' *)
(* @SYMFILEFLAGS := '2048' *)
FUNCTION_BLOCK INC_DEC
VAR_INPUT
	CHa : BOOL;
	CHb : BOOL;
	RST : BOOL;
END_VAR
VAR_OUTPUT
	dir : BOOL;
	cnt : INT;
END_VAR
VAR
	edgea : BOOL;
	clk: BOOL;
	clka: BOOL;
	clkb: BOOL;
	edgeb: BOOL;
	axb: BOOL;
END_VAR

(*
	version 1.0	4 aug 2006
	programmer 	oscat
	tested BY		oscat

incremental decoder with quadruple accuracy.
2 pulses for each channel are created for each directional pulse.
*)
(* @END_DECLARATION := '0' *)
axb := cha XOR chb;

(* create pulses for channel a *)
clka := cha XOR edgea;
edgea := cha;

clkb := chb XOR edgeb;
edgeb := chb;

(* create pulses for both channels *)
clk := clka OR clkb;

(* set the direction output *)
IF axb AND clka THEN dir := TRUE; END_IF;
IF axb AND clkb THEN dir := FALSE; END_IF;

(* increment or decrement the counter *)
IF clk AND dir THEN cnt := cnt + 1; END_IF;
IF clk AND NOT dir THEN cnt := cnt -1; END_IF;

(* reset the counter if rst active *)
IF rst THEN cnt := 0; END_IF;

END_FUNCTION_BLOCK

(* @NESTEDCOMMENTS := 'Yes' *)
(* @PATH := '\/Engineering\/automation' *)
(* @OBJECTFLAGS := '0, 8' *)
(* @SYMFILEFLAGS := '2048' *)
FUNCTION_BLOCK INTERLOCK
VAR_INPUT
	I1, I2 : BOOL;
	TL : TIME;
END_VAR
VAR_OUTPUT
	Q1, Q2 : BOOL;
END_VAR
VAR
	T1, T2 : TOF;
END_VAR

(*
version 1.0	28 sep 2007
programmer 	hugo
tested by		tobias

INTERLOCK has two inputs I1 and I2 which drive the corresponding outputs Q1 and Q2.
the inputs signals lock each other out and therfore I1 can only drive Q1 when I2 is Low and vice versa.
The input TL specifies a dead time between two outputs can become active.
an output can only become active when the other output was not active for the time TL.

*)
(* @END_DECLARATION := '0' *)
(* the input signal have a run delay to lockout the other input *)
T1(IN := I1, PT := TL);
T2(IN := I2, PT := TL);

Q1 := I1 AND NOT t2.Q;
Q2 := I2 AND NOT t1.Q;

(* revision history

hm	28 sep 2007		rev 1.0
	original version

*)
END_FUNCTION_BLOCK

(* @NESTEDCOMMENTS := 'Yes' *)
(* @PATH := '\/Engineering\/automation' *)
(* @OBJECTFLAGS := '0, 8' *)
(* @SYMFILEFLAGS := '2048' *)
FUNCTION_BLOCK INTERLOCK_4
VAR_INPUT (* CONSTANT *)
END_VAR
VAR_INPUT
	I0 : BOOL;
	I1 : BOOL;
	I2 : BOOL;
	I3 : BOOL;
	E : BOOL;
	MODE : INT;

END_VAR
VAR_OUTPUT
	OUT : BYTE;
	TP : BOOL;
END_VAR
VAR
	in: BYTE;
	last: BYTE;
	old: BYTE;
	lmode: INT;
END_VAR

(*
version 1.1	14. mar. 2009
programmer 	hugo
tested by		oscat

INTERLOCK_4 detects one of 4 switches and delivers the number of the switch pressed on the output out
a output tp is true for one cycle if the output has changed.
a setup variable MODE selects between 3 different modes:
MODE = 0, any input active will disable all other inputs
MODE = 1, the input with the highest number will be acepted
mode = 2, the input last pressed will disable all others

*)
(* @END_DECLARATION := '0' *)
(* check if enable is active *)
IF E THEN
(* reset all vars when there is a mode change on thy fly *)
	IF mode <> lmode THEN
		out := 0;
		last := 0;
		old := 0;
		lmode := mode;
	END_IF;
	(* load inputs into in *)
	in.0 := I0;
	in.1 := I1;
	in.2 := I2;
	in.3 := I3;
	(* only execute when there is any change *)
	IF in <> last THEN
		(* only execute when inputs have chages state *)
		CASE mode OF
			0:	(* output directly display inputs as bits in byte out *)
				out := in;

			1:	(* the input with the highest number will be acepted *)
				IF in.3 THEN out := 8;
				ELSIF in.2 THEN out := 4;
				ELSIF in.1 THEN out := 2;
				ELSE out := in;
				END_IF;

			2:	(* input last pressed will be displayed only *)
				last := ((in XOR last) AND in);
				IF last.3 THEN out := 8;
				ELSIF last.2 THEN out := 4;
				ELSIF last.1 THEN out := 2;
				ELSE out := last;
				END_IF;

			3:	(* any input active will disable all other inputs *)
				IF (out AND in) = 0 THEN
					IF in.3 THEN out := 8;
					ELSIF in.2 THEN out := 4;
					ELSIF in.1 THEN out := 2;
					ELSE out := in;
					END_IF;
				END_IF;

		END_CASE;
		last := in;
	END_IF;
	tp := out <> old;
	old := out;
ELSE
	out := 0;
	last := 0;
	old := 0;
	lmode := 0;
	tp := FALSE;
END_IF;

(* revision history
hm	24. oct 2008	rev 1.0
	original version

hm	14. mar. 2009	rev 1.1
	replaced double assignments

*)
END_FUNCTION_BLOCK

(* @NESTEDCOMMENTS := 'Yes' *)
(* @PATH := '\/Engineering\/automation' *)
(* @OBJECTFLAGS := '0, 8' *)
(* @SYMFILEFLAGS := '2048' *)
FUNCTION MANUAL : BOOL
VAR_INPUT
	IN : BOOL;
	ON : BOOL;
	OFF : BOOL;
END_VAR

(*
version 1.0	21. nov. 2008
programmer 	hugo
tested by	oscat

MANUAL is a manual override for digital signals.
when on and off = FALSE, the output follows IN.
ON = TRUE forces the output high, and OFF = TRUE forces the output low.

*)
(* @END_DECLARATION := '0' *)
MANUAL := NOT OFF AND (IN OR ON);

(* revision history
hm	21. nov 2008	rev 1.0
	original version

*)
END_FUNCTION

(* @NESTEDCOMMENTS := 'Yes' *)
(* @PATH := '\/Engineering\/automation' *)
(* @OBJECTFLAGS := '0, 8' *)
(* @SYMFILEFLAGS := '2048' *)
FUNCTION_BLOCK MANUAL_1
VAR_INPUT
	IN : BOOL;
	MAN : BOOL;
	M_I : BOOL;
	SET0 : BOOL;
	RST : BOOL;
END_VAR
VAR_OUTPUT
	Q : BOOL;
	STATUS : BYTE;
END_VAR
VAR
	S_edge : BOOL;
	r_edge : BOOL;
	edge: BOOL;
END_VAR

(*
version 1.2	14. mar. 2009
programmer 	hugo
tested by		oscat

MANUAL_1 is a manual override for digital signals.
When MAN = FALSE, the output follows IN and when MAN = TRUE the Output follows M_I.

*)
(* @END_DECLARATION := '0' *)
IF NOT man THEN
	Q := IN;
	STATUS := 100;
	edge := FALSE;
ELSIF NOT s_edge AND set0 THEN
	Q := TRUE;
	edge := TRUE;
	status := 101;
ELSIF NOT r_edge AND rst THEN
	Q := FALSE;
	edge := TRUE;
	status := 102;
ELSIF NOT edge THEN
	Q := M_I;
	status := 103;
END_IF;

(* remember levels of manual signals *)
s_edge := SET0;
r_edge := RST;

(* revision history
hm	17. jun 2008	rev 1.0
	original version

hm	17. oct 2008	rev 1.1
	deleted unnecessary variable m_edge

hm	14. mar. 2009	rev 1.2
	replaced double assignments

*)
END_FUNCTION_BLOCK

(* @NESTEDCOMMENTS := 'Yes' *)
(* @PATH := '\/Engineering\/automation' *)
(* @OBJECTFLAGS := '0, 8' *)
(* @SYMFILEFLAGS := '2048' *)
FUNCTION_BLOCK MANUAL_2
VAR_INPUT
	IN : BOOL;
	ENA : BOOL;
	ON : BOOL;
	OFF : BOOL;
	MAN : BOOL;
END_VAR
VAR_OUTPUT
	Q : BOOL;
	STATUS : BYTE;
END_VAR

(*
version 1.0	22. sep. 2008
programmer 	hugo
tested by	oscat

MANUAL_2 is a manual override for boolean signals.
it has static force high and low as well as a manual input.

*)
(* @END_DECLARATION := '0' *)
IF ena THEN
	IF NOT ON AND NOT OFF THEN
		Q := IN;
		STATUS := 100;
	ELSIF on AND NOT off THEN
		Q := TRUE;
		STATUS := 101;
	ELSIF NOT on AND off THEN
		q := FALSE;
		STATUS := 102;
	ELSE
		Q := MAN;
		STATUS := 103;
	END_IF;
ELSE
	Q := FALSE;
	STATUS := 104;
END_IF;

(* revision history
hm	22. sep. 2008		rev 1.0
	original version

*)
END_FUNCTION_BLOCK

(* @NESTEDCOMMENTS := 'Yes' *)
(* @PATH := '\/Engineering\/automation' *)
(* @OBJECTFLAGS := '0, 8' *)
(* @SYMFILEFLAGS := '2048' *)
FUNCTION_BLOCK MANUAL_4
VAR_INPUT
	I0, I1, I2, I3 : BOOL;
	MAN : BOOL;
	STP : BOOL;
	M0, M1, M2, M3 : BOOL;
END_VAR
VAR_OUTPUT
	Q0, Q1, Q2, Q3 : BOOL;
	STATUS : BYTE;
END_VAR
VAR
	edge: BOOL;
	pos : INT;
	tog: BOOL;
END_VAR

(*
version 1.0	17. jun 2008
programmer 	hugo
tested by	oscat

MANUAL_4 is a manual override for digital signals.
When MAN = FALSE, the output follows IN and when MAN = TRUE the Output follows M_I.

*)
(* @END_DECLARATION := '0' *)
IF man THEN
	IF NOT TOG THEN
		Q0 := M0;
		Q1 := M1;
		Q2 := M2;
		Q3 := M3;
		STATUS := 101;
	END_IF;
	IF STP AND NOT edge THEN
		tog := TRUE;
		CASE pos OF
			0:	Q0 := TRUE;
				Q1 := FALSE;
				Q2 := FALSE;
				Q3 := FALSE;
				STATUS := 110;
			1:	Q0 := FALSE;
				Q1 := TRUE;
				Q2 := FALSE;
				Q3 := FALSE;
				STATUS := 111;
			2:	Q0 := FALSE;
				Q1 := FALSE;
				Q2 := TRUE;
				Q3 := FALSE;
				STATUS := 112;
			3:	Q0 := FALSE;
				Q1 := FALSE;
				Q2 := FALSE;
				Q3 := TRUE;
				STATUS := 113;
		END_CASE;
		pos := INC(pos,1,3);
	END_IF;
ELSE
	Q0 := I0;
	Q1 := I1;
	Q2 := I2;
	Q3 := I3;
	STATUS := 100;
	tog := FALSE;
	pos := 0;
END_IF;

(* remember status of stp *)
edge := STP;

(* revision history
hm	17. jun 2008		rev 1.0
	original version

*)
END_FUNCTION_BLOCK

(* @NESTEDCOMMENTS := 'Yes' *)
(* @PATH := '\/Engineering\/automation' *)
(* @OBJECTFLAGS := '0, 8' *)
(* @SYMFILEFLAGS := '2048' *)
FUNCTION_BLOCK PARSET
VAR_INPUT
	A0, A1 : BOOL;
END_VAR
VAR_INPUT (* CONSTANT *)
	X01, X02, X03, X04 : REAL;
	X11, X12, X13, X14 : REAL;
	X21, X22, X23, X24 : REAL;
	X31, X32, X33, X34 : REAL;
	TC : TIME;
END_VAR
VAR_OUTPUT
	P1, P2, P3, P4 : REAL;
END_VAR
VAR
	X : ARRAY[0..3,1..4] OF REAL;
	S1, S2, S3, S4 : REAL;
	tx, last : DWORD;
	start : BOOL;
	set0 : BYTE;
	init: BOOL;
END_VAR

(*
version 1.1	16. mar. 2008
programmer 	hugo
tested by		tobias

parset selects on of 4 parameter sets adressed by the inputs A0 and A1. if TC is specified, the change of the outputs
is ramped by the time tc
*)

(* @END_DECLARATION := '0' *)
(* read system_time *)
tx := T_PLC_MS();

(* init sequence *)
IF NOT init THEN
	set0.0 := NOT A0;
	init := TRUE;
	X[0,1] := X01;
	X[0,2] := X02;
	X[0,3] := X03;
	X[0,4] := X04;
	X[1,1] := X11;
	X[1,2] := X12;
	X[1,3] := X13;
	X[1,4] := X14;
	X[2,1] := X21;
	X[2,2] := X22;
	X[2,3] := X23;
	X[2,4] := X24;
	X[3,1] := X31;
	X[3,2] := X32;
	X[3,3] := X33;
	X[3,4] := X34;
	P1 := X01;
	P2 := X02;
	P3 := X03;
	P4 := X04;
END_IF;

(* check for input change *)
IF (A0 XOR set0.0) OR (A1 XOR set0.1) THEN
	(* a new set is selected *)
	set0.0 := A0;
	set0.1 := A1;
	IF tc > t#0s THEN
		start := TRUE;
		last := tx;
		(* save the step speed for the output changes in S *)
		S1 := (X[set0,1] - P1)/DWORD_TO_REAL(TIME_TO_DWORD(tc));
		S2 := (X[set0,2] - P2)/DWORD_TO_REAL(TIME_TO_DWORD(tc));
		S3 := (X[set0,3] - P3)/DWORD_TO_REAL(TIME_TO_DWORD(tc));
		S4 := (X[set0,4] - P4)/DWORD_TO_REAL(TIME_TO_DWORD(tc));
	END_IF;
ELSIF start AND tx - last < TIME_TO_DWORD(tc) THEN
	(* ramp the outputs to the new value *)
	P1 := X[set0,1] - S1 * DWORD_TO_REAL(TIME_TO_DWORD(Tc) - tx + last);
	P2 := X[set0,2] - S2 * DWORD_TO_REAL(TIME_TO_DWORD(Tc) - tx + last);
	P3 := X[set0,3] - S3 * DWORD_TO_REAL(TIME_TO_DWORD(Tc) - tx + last);
	P4 := X[set0,4] - S4 * DWORD_TO_REAL(TIME_TO_DWORD(Tc) - tx + last);
ELSE
	(* make sure outputs match the correct set values *)
	start := FALSE;
	P1 := X[set0,1];
	P2 := X[set0,2];
	P3 := X[set0,3];
	P4 := X[set0,4];
END_IF;

(* revision history
hm	2.11.2007		rev 1.0
	original version

hm	16. mar. 2008	rev 1.1
	added type conversions to avoid warnings under codesys 3.0

*)

END_FUNCTION_BLOCK

(* @NESTEDCOMMENTS := 'Yes' *)
(* @PATH := '\/Engineering\/automation' *)
(* @OBJECTFLAGS := '0, 8' *)
(* @SYMFILEFLAGS := '2048' *)
FUNCTION_BLOCK PARSET2
VAR_INPUT
	X : REAL;
END_VAR
VAR_INPUT (* CONSTANT *)
	X01, X02, X03, X04 : REAL;
	X11, X12, X13, X14 : REAL;
	X21, X22, X23, X24 : REAL;
	X31, X32, X33, X34 : REAL;
	L1, L2, L3 : REAL;
	TC : TIME;
END_VAR
VAR_OUTPUT
	P1,P2,P3,P4 : REAL;
END_VAR
VAR
	Pset : parset;
	init: BOOL;
END_VAR

(*
version 1.0	3 nov 2007
programmer 	hugo
tested by	tobias

parset2 selects on of 4 parameter sets depending on the value of X. if TC is specified, the change of the outputs
is ramped by the time TC
*)

(* @END_DECLARATION := '0' *)
(* init sequence *)
IF NOT init THEN
	init := TRUE;
	pset(TC:=TC, X01:=X01, X02:=X02, X03:=X03, X04:=X04, X11:=X11, X12:=X12, X13:=X13, X14:=X14, X21:=X21, X22:=X22, X23:=X23, X24:=X24, X31:=X31, X32:=X32, X33:=X33, X34:=X34);
END_IF;
IF ABS(X) < L1 THEN
	pset(A0 := FALSE, A1 := FALSE);
ELSIF ABS(X) < L2 THEN
	pset(A0 := TRUE, A1 := FALSE);
ELSIF ABS(x) < L3 THEN
	pset(A0 := FALSE, A1 := TRUE);
ELSE
	pset(A0 := TRUE, A1 := TRUE);
END_IF;
P1 := pset.P1;
P2 := pset.P2;
P3 := pset.P3;
P4 := pset.P4;

(* revision history
hm		3.11.2007		rev 1.0
	original version

*)

END_FUNCTION_BLOCK

(* @NESTEDCOMMENTS := 'Yes' *)
(* @PATH := '\/Engineering\/automation' *)
(* @OBJECTFLAGS := '0, 8' *)
(* @SYMFILEFLAGS := '2048' *)
FUNCTION_BLOCK SIGNAL
VAR_INPUT
	IN : BOOL;
	SIG : BYTE;
	TS : TIME;
END_VAR
VAR_OUTPUT
	Q : BOOL;
END_VAR
VAR
	tx: DWORD;
	step: BYTE;
END_VAR
VAR CONSTANT
	one : BYTE := 1;
END_VAR

(*
version 1.0	13 dec 2007
programmer 	hugo
tested by		tobias

this function generates an output signal according to a bit pattern SIG.
the patter is shifted to the output in time steps of TS.
ts defaults to 128 ms if not specified.
*)

(* @END_DECLARATION := '0' *)
IF in THEN
	(* an alarm is present read system time first *)
	tx := T_PLC_MS();
	(* calculate the step counter which is the lowest 3 bits of (time / ts) *)
	IF ts > t#0s THEN
		step := DWORD_TO_BYTE(tx / TIME_TO_DWORD(ts) AND 16#0000_0007);
	ELSE
		step := DWORD_TO_BYTE(SHR(tx,7) AND 16#0000_0007);
	END_IF;
	(* convert the value 0-7 in step into one bit only (bit 0-7) *)
	step := SHL(one,step);
	(* generate the output signal *)
	Q := (step AND sig) > 0;
ELSE
	Q := FALSE;
END_IF;

(* revision history
hm	13.12.2007		rev 1.0
	original version

*)
END_FUNCTION_BLOCK

(* @NESTEDCOMMENTS := 'Yes' *)
(* @PATH := '\/Engineering\/automation' *)
(* @OBJECTFLAGS := '0, 8' *)
(* @SYMFILEFLAGS := '2048' *)
FUNCTION_BLOCK SIGNAL_4
VAR_INPUT
	IN1 : BOOL;
	IN2 : BOOL;
	IN3 : BOOL;
	IN4 : BOOL;
	TS : TIME;
END_VAR
VAR_INPUT (* CONSTANT *)
	S1 : BYTE := 2#1111_1111;
	S2 : BYTE := 2#1111_0000;
	S3 : BYTE := 2#1010_1010;
	S4 : BYTE := 2#1010_0000;
END_VAR
VAR_OUTPUT
	Q : BOOL;
END_VAR
VAR
	sig : SIGNAL;
END_VAR

(*
version 1.0	13 dec 2007
programmer 	hugo
tested by		tobias

this function generates one out of 4 signals specified by bit patterns S1 .. S4.
the selected pattern will be shifted with the step time TS.
In1 has higher priority then In2 which has higher priority then IN3 and in4 has the lowest priority.
ts defaults to 128 ms if not specified.
*)

(* @END_DECLARATION := '0' *)
(* an alarm is present read system time first *)
(* check if an alarm is present if yes set sig to the alarm pattern otherwise exit the routine *)
IF in1 THEN
	sig(in := TRUE, sig := s1, TS := TS);
ELSIF in2 THEN
	sig(in := TRUE, sig := s2, TS := TS);
ELSIF in3 THEN
	sig(in := TRUE, sig := s3, TS := TS);
ELSIF in4 THEN
	sig(in := TRUE, sig := s4, TS := TS);
ELSE
	sig(in := FALSE);
END_IF;

(* set the output *)
Q := sig.Q;

(* revision history
hm	13.12.2007		rev 1.0
	original version

*)

END_FUNCTION_BLOCK

(* @NESTEDCOMMENTS := 'Yes' *)
(* @PATH := '\/Engineering\/automation' *)
(* @OBJECTFLAGS := '0, 8' *)
(* @SYMFILEFLAGS := '2048' *)
FUNCTION_BLOCK SRAMP
VAR_INPUT
	X : REAL;
	A_UP : REAL;
	A_DN :REAL;
	VU_MAX : REAL;
	VD_MAX : REAL;
	LIMIT_HIGH : REAL;
	LIMIT_LOW : REAL;
	RST : BOOL;
END_VAR
VAR_OUTPUT
	Y : REAL;
	V : REAL;
END_VAR
VAR
	cycle_time : TC_S;
	init: BOOL;
END_VAR

(*
	version 1.1	11. mar. 2009
	programmer 	hugo
	tested by		tobias

RAMPS generates output signal which are slew rate and acceleration controlled.

*)
(* @END_DECLARATION := '0' *)
(* read the system_time in microseconds *)
cycle_time();

(* assure range of inputs *)
A_up := MAX(0.0, A_UP);
A_dn := MIN(0.0, A_dn);
VU_max := MAX(0.0, VU_max);
VD_max := MIN(0.0, VD_MAX);

(* calculate the output offset *)
IF rst OR NOT init THEN
	init := TRUE;
	Y := 0.0;
	V := 0.0;
ELSIF X = Y THEN
	v := 0.0;
ELSIF X > Y THEN
	(* output is too low >> ramp up and brake at the end *)
	(* accelerate the speed and limit to vu_max *)
	v := MIN(v + A_UP * cycle_time.TC, vu_max);
	(* calculate the max speed to be able to brake and select the lowest *)
	v := MIN(SQRT((Y-X) * 2.0 * A_DN), v);
	(* calculate the output and obey limits *)
	y := LIMIT(limit_low, y + MIN(v * cycle_time.TC, X-Y), limit_high);
ELSIF X < Y THEN
	(* output is too high >> ramp dn and brake at the end *)
	(* accelerate the speed and limit to vd_max *)
	v := MAX(v + A_DN * cycle_time.TC, vd_max);
	(* calculate the max speed to be able to brake and select the lowest *)
	v := MAX(-SQRT((Y-X) * 2.0 * A_UP), v);
	(* calculate the output and obey limits *)
	y := LIMIT(limit_low, y + MAX(v * cycle_time.TC, X-Y), limit_high);
END_IF;

(* revision history
hm	13. mar. 2008	rev 1.0
	original version

hm	11. mar. 2009	rev 1.1
	real constants updated to new systax using dot

*)

END_FUNCTION_BLOCK

(* @NESTEDCOMMENTS := 'Yes' *)
(* @PATH := '\/Engineering\/automation' *)
(* @OBJECTFLAGS := '0, 8' *)
(* @SYMFILEFLAGS := '2048' *)
FUNCTION_BLOCK TUNE
VAR_INPUT
	SET0 : BOOL;
	SU, SD : BOOL;
	RST : BOOL;
END_VAR
VAR_INPUT (* CONSTANT *)
	SS : REAL := 0.1;
	Limit_L : REAL;
	LIMIT_H : REAL := 100.0;
	RST_val : REAL;
	SET_val : REAL := 100.0;
	T1 : TIME := T#500ms;
	T2 : TIME := T#2s;
	S1 : REAL := 2.0;
	S2 : REAL := 10.0;
END_VAR
VAR_OUTPUT
	Y : REAL;
END_VAR
VAR
	tx : DWORD;
	start, start2 : DWORD;
	state : INT;
	in : BOOL;
	step : REAL;
	SPEED : REAL;
	Y_start : REAL;
	Y_start2: REAL;
END_VAR

(*
version 1.2	11. mar. 2009
programmer 	hugo
tested by		tobias

tune generates an output signal which is set by input switches.
up to 4 switsches can be used to tune the signal up or down.

*)

(* @END_DECLARATION := '0' *)
(* read system time *)
tx := T_PLC_MS();

IF rst THEN
	Y := RST_val;
	state := 0;
ELSIF set0 THEN
	Y := SET_val;
	state := 0;
ELSIF state > 0 THEN
	(* key has been pushed state machine operating *)
	(* first read the correct input *)
	IF state = 1 THEN
		(* step up *)
		in := su;
	ELSE
		(* step down *)
		in := sd;
	END_IF;
	(* check for single step operation *)
	IF NOT in AND tx - start <= TIME_TO_DWORD(T1) THEN
		Y := Y_start + step;
		state := 0;
	(* check if fast ramp needs to be generated *)
	ELSIF in AND tx - start >= TIME_TO_DWORD(T2) THEN
		Y := Y_start2 + DWORD_TO_REAL(tx - start2) * s2 / speed;
	(* check if slow ramp needs to be generated *)
	ELSIF in AND tx - start >= TIME_TO_DWORD(T1) THEN
		Y := Y_start + DWORD_TO_REAL(tx - start - TIME_TO_DWORD(T1)) * S1 / speed;
		start2 := tx;
		Y_start2 := Y;
	ELSIF NOT in THEN
		state := 0;
	END_IF;
ELSIF su THEN
	(* slow step up *)
	state := 1;
	start := tx;
	step := ss;
	speed := 1000.0;
	Y_start := Y;
ELSIF sd THEN
	(* slow step down *)
	state := 2;
	start := tx;
	step := -ss;
	speed := -1000.0;
	Y_start := Y;
END_IF;

(* make sure output does not exceed limits *)
Y := LIMIT(LIMIT_L, Y, LIMIT_H);

(* revision history
hm	3.11.2007		rev 1.0
	original version

hm	16. mar. 2008	rev 1.1
	added type conversions to avoid warnings under codesys 3.0

hm	11. mar. 2009	rev 1.2
	real constants updated to new systax using dot

*)
END_FUNCTION_BLOCK

(* @NESTEDCOMMENTS := 'Yes' *)
(* @PATH := '\/Engineering\/automation' *)
(* @OBJECTFLAGS := '0, 8' *)
(* @SYMFILEFLAGS := '2048' *)
FUNCTION_BLOCK TUNE2
VAR_INPUT
	SET0 : BOOL;
	SU, SD : BOOL;
	FU, FD : BOOL;
	RST : BOOL;
END_VAR
VAR_INPUT (* CONSTANT *)
	SS : REAL := 0.1;
	FS : REAL := 5.0;
	Limit_L : REAL;
	LIMIT_H : REAL := 100.0;
	RST_val : REAL;
	SET_val : REAL := 100.0;
	TR : TIME := T#500ms;
	S1 : REAL := 2.0;
	S2 : REAL := 10.0;
END_VAR
VAR_OUTPUT
	Y : REAL;
END_VAR
VAR
	tx : DWORD;
	start : DWORD;
	state : INT;
	in : BOOL;
	step : REAL;
	SPEED : REAL;
	Y_start : REAL;
END_VAR

(*
version 1.2	11. mar. 2009
programmer 	hugo
tested by		tobias

tune2 generates an output signal which is set by input switches.
up to 4 switsches can be used to tune the signal up or down.

*)

(* @END_DECLARATION := '0' *)
(* read system time *)
tx := T_PLC_MS();

IF rst THEN
	Y := RST_val;
	state := 0;
ELSIF set0 THEN
	Y := SET_val;
	state := 0;
ELSIF state > 0 THEN
	(* key has been pushed state machine operating *)
	(* first read the correct input *)
	CASE state OF
		1 :	(* slow up *)
			in := su;
		2 :	(* slow down *)
			in := sd;
		3 :	(* fast up *)
			in := fu;
		4 :	(* fast down *)
			in := fd;
	END_CASE;
	(* check for single step operation *)
	IF NOT in AND tx - start <= TIME_TO_DWORD(TR) THEN
		Y := Y_start + step;
		state := 0;
	(* check if ramp needs to be generated *)
	ELSIF in AND tx - start >= TIME_TO_DWORD(TR) THEN
		Y := Y_start + DWORD_TO_REAL(tx - start - TIME_TO_DWORD(TR)) * speed;
	ELSIF NOT in THEN
		state := 0;
	END_IF;
ELSIF su THEN
	(* slow step up *)
	state := 1;
	start := tx;
	step := ss;
	speed := s1 * 1.0E-3;
	Y_start := Y;
ELSIF sd THEN
	(* slow step down *)
	state := 2;
	start := tx;
	step := -ss;
	speed := -s1 * 1.0E-3;
	Y_start := Y;
ELSIF fu THEN
	(* fast step up *)
	state := 3;
	start := tx;
	step := fs;
	speed := s2 * 1.0E-3;
	y_start := Y;
ELSIF fd THEN
	(* fast step down *)
	state := 4;
	start := tx;
	step := -fs;
	speed := -s2 * 1.0E-3;
	y_start := Y;
END_IF;

(* make sure output does not exceed limits *)
Y := LIMIT(LIMIT_L, Y, LIMIT_H);

(* revision history
hm	3.11.2007		rev 1.0
	original version

hm	16. 3. 2008	rev 1.1
	added type conversions to avoid warnings in codesys 3.0
	improved performance

hm	11. mar. 2009	rev 1.2
	real constants updated to new systax using dot

*)
END_FUNCTION_BLOCK

(* @NESTEDCOMMENTS := 'Yes' *)
(* @PATH := '\/Engineering\/control' *)
(* @OBJECTFLAGS := '0, 8' *)
(* @SYMFILEFLAGS := '2048' *)
FUNCTION BAND_B : BYTE
VAR_INPUT
	X : BYTE;
	B : BYTE;
END_VAR

(*
version 1.0	21. Nov. 2008
programmer 	hugo
tested by	oscat

BAND_B will limit X to B <= X <= 255-B. while X < B the resulkt will be 0 and while X > 255-B the output will be 255
otherwise the result = X.

*)
(* @END_DECLARATION := '0' *)
IF X < B THEN
	BAND_B := 0;
ELSIF X > BYTE#255-B THEN
	BAND_B := 255;
ELSE
	BAND_B := X;
END_IF;

(* revision history
hm	21. nov. 2008	rev 1.0
	original version

*)

END_FUNCTION

(* @NESTEDCOMMENTS := 'Yes' *)
(* @PATH := '\/Engineering\/control' *)
(* @OBJECTFLAGS := '0, 8' *)
(* @SYMFILEFLAGS := '2048' *)
FUNCTION_BLOCK CONTROL_SET1
VAR_INPUT
	Kt : REAL;
	Tt : REAL;
	PI : BOOL;
	PID : BOOL;
END_VAR
VAR_INPUT (* CONSTANT *)
	P_K : REAL := 0.5;
	PI_K : REAL := 0.45;
	PI_TN : REAL := 0.83;
	PID_K : REAL := 0.6;
	PID_TN : REAL := 0.5;
	PID_TV : REAL := 0.125;
END_VAR
VAR_OUTPUT
	KP : REAL;
	TN : REAL;
	TV : REAL;
	KI : REAL;
	KD : REAL;
END_VAR

(*
version 1.1	11. mar. 2009
programmer 	hugo
tested by		tobias

takahashi calculates controller parameters for P, PI and PID controllers based on the ziegler nichols method.

*)

(* @END_DECLARATION := '0' *)
IF pi AND PID THEN
	KP := 0.0;
	TN := 0.0;
	TV := 0.0;
ELSIF PID THEN
	KP := PID_K * Kt;
	TN := PID_TN * Tt;
	TV := PID_TV * Tt;
ELSIF PI THEN
	KP := PI_K * Kt;
	TN := PI_TN * Tt;
ELSE
	KP := P_K * Kt;
END_IF;

(* KI and KD are calculated *)
IF tn > 0.0 THEN KI := KP / TN; ELSE KI := 0.0; END_IF;
KD := KP * TV;

(* revision history
hm	4. nov 2007	rev 1.0
	original version

hm	11. mar. 2009	rev 1.1
	real constants updated to new systax using dot

*)
END_FUNCTION_BLOCK

(* @NESTEDCOMMENTS := 'Yes' *)
(* @PATH := '\/Engineering\/control' *)
(* @OBJECTFLAGS := '0, 8' *)
(* @SYMFILEFLAGS := '2048' *)
FUNCTION_BLOCK CONTROL_SET2
VAR_INPUT
	KS : REAL;
	TU : REAL;
	TG : REAL;
	PI : BOOL;
	PID : BOOL;
END_VAR
VAR_INPUT (* CONSTANT *)
	P_K : REAL := 1.0;
	PI_K : REAL := 0.9;
	PI_TN : REAL := 3.33;
	PID_K : REAL := 1.2;
	PID_TN : REAL := 2.0;
	PID_TV : REAL := 0.5;
END_VAR
VAR_OUTPUT
	KP : REAL;
	TN : REAL;
	TV : REAL;
	KI : REAL;
	KD : REAL;
END_VAR
VAR
	TX : REAL;
END_VAR

(*
version 1.1	11. mar. 2009
programmer 	hugo
tested by		tobias

takahashi calculates controller parameters for P, PI and PID controllers based on the ziegler nichols method.

*)

(* @END_DECLARATION := '0' *)
IF TU > 0.0 AND KS > 0.0 THEN TX := TG / TU / KS; END_IF;
IF pi AND PID THEN
	KP := 0.0;
	TN := 0.0;
	TV := 0.0;
ELSIF PID THEN
	KP := PID_K * TX;
	TN := PID_TN * TU;
	TV := PID_TV * TU;
ELSIF PI THEN
	KP := PI_K * TX;
	TN := PI_TN * TU;
ELSE
	KP := P_K * TX;
END_IF;

(* KI and KD are calculated *)
IF TN > 0.0 THEN KI := KP / TN; ELSE KI := 0.0; END_IF;
KD := KP * TV;

(* revision history
hm	4. nov 2007	rev 1.0
	original version

hm	11. mar. 2009	rev 1.1
	real constants updated to new systax using dot

*)
END_FUNCTION_BLOCK

(* @NESTEDCOMMENTS := 'Yes' *)
(* @PATH := '\/Engineering\/control' *)
(* @OBJECTFLAGS := '0, 8' *)
(* @SYMFILEFLAGS := '2048' *)
FUNCTION CTRL_IN : REAL
VAR_INPUT
	SET_POINT, ACTUAL, NOISE : REAL;
END_VAR

(*
version 1.0	2. jun 2008
programmer 	hugo
tested by		tobias

*)

(* @END_DECLARATION := '0' *)
(* calculate the process error DIFF *)
CTRL_IN := DEAD_ZONE(SET_POINT - ACTUAL, NOISE);

(* revision history
hm 	2. jun. 2008 	rev 1.0
	original version

*)
END_FUNCTION

(* @NESTEDCOMMENTS := 'Yes' *)
(* @PATH := '\/Engineering\/control' *)
(* @OBJECTFLAGS := '0, 8' *)
(* @SYMFILEFLAGS := '2048' *)
FUNCTION_BLOCK CTRL_OUT
VAR_INPUT
	CI, OFFSET, MAN_IN, LIM_L, LIM_H : REAL;
	MANUAL : BOOL;
END_VAR
VAR_OUTPUT
	Y : REAL;
	LIM : BOOL;
END_VAR

(*
version 1.1	5. nov 2008
programmer 	hugo
tested by	oscat

*)

(* @END_DECLARATION := '0' *)
Y := SEL(MANUAL, CI, MAN_IN) + OFFSET;

(* Limit the output *)
IF Y > LIM_L AND Y < LIM_H THEN
	LIM := FALSE;
ELSE
	Y := LIMIT(LIM_L, Y, LIM_H);
	LIM := TRUE;
END_IF;

(* revision history
hm 	2. jun. 2008 	rev 1.0
	original version

hm	5. nov. 2008	rev 1.1
	optimized code
*)
END_FUNCTION_BLOCK

(* @NESTEDCOMMENTS := 'Yes' *)
(* @PATH := '\/Engineering\/control' *)
(* @OBJECTFLAGS := '0, 8' *)
(* @SYMFILEFLAGS := '2048' *)
FUNCTION_BLOCK CTRL_PI
VAR_INPUT
	ACT, SET0, SUP, OFS, M_I : REAL;
	MAN : BOOL;
	RST : BOOL;
	KP : REAL := 1.0;
	KI : REAL := 1.0;
	LL : REAL := -1000.0;
	LH : REAL := 1000.0;
END_VAR
VAR_OUTPUT
	Y : REAL;
	DIFF : REAL;
	LIM : BOOL;
END_VAR
VAR
	pi : FT_PIWL;
	co : CTRL_OUT;
END_VAR

(*
version 2.0	30. jun 2008
programmer 	hugo
tested by	oscat

FT_PI is a PI controller with manual functionality.
The PID controller works according to the fomula Y = e *(KP+ KI * INTEG(e) ) + offset, while e = set_point - actual.
a rst will reset all internal data, while a switch to manual will cause the controller to follow the function Y = manual_in + offset.
limit_h and Limit_l set the possible output range of Y.
the output flags lim will signal that the output limits are active and overflow will signal that the integrator has reached its limits.

since rev 1.1 the "trapezregel is used for more accuracy.
rev 1.2 added selective integratin which means the integrative component is only active within a small range of the target value
this avoids the integrator to go to limits while an input setpoint change happened and is only causing overshoots.
the int_band is by default 100 which means the int is active all the time and if set to for example to 0.1 the integrator is only active
while the input is between 0.9 and 1.1 of the set_point value.

default values for KP = 1, TN = 1, TV = 1, LIMIT_L = -1000, LIMIT_H = +1000.
*)

(* @END_DECLARATION := '0' *)
DIFF := CTRL_IN(SET0, ACT, SUP);
pi(in := DIFF, kp := KP, ki := KI, lim_l := LL, lim_h := LH, rst := RST);
co(ci := pi.Y, OFFSET := OFS, man_in := M_I, lim_l := LL, lim_h := LH, MANUAL := MAN);
Y := co.Y;
LIM := co.LIM;

(* revision history
hm 	31.10.2007 		rev 1.0
	original version

hm	3.11.2007		rev 1.1
	added noise input to filter noise
	added output diff
	set limit output false when output is within limits
	overfolw was not set correctly

hm	5. jan 2008		rev 1.2
	improved performance

hm	20. jun. 2008	rev 2.0
	rewritten using new modular approach

*)
END_FUNCTION_BLOCK

(* @NESTEDCOMMENTS := 'Yes' *)
(* @PATH := '\/Engineering\/control' *)
(* @OBJECTFLAGS := '0, 8' *)
(* @SYMFILEFLAGS := '2048' *)
FUNCTION_BLOCK CTRL_PID
VAR_INPUT
	ACT, SET0, SUP, OFS, M_I : REAL;
	MAN : BOOL;
	RST : BOOL;
	KP : REAL := 1.0;
	TN : REAL := 1.0;
	TV : REAL := 1.0;
	LL : REAL := -1000.0;
	LH : REAL := 1000.0;
END_VAR
VAR_OUTPUT
	Y : REAL;
	DIFF : REAL;
	LIM : BOOL;
END_VAR
VAR
	pid : FT_PIDWL;
	co : CTRL_OUT;
END_VAR

(*
version 2.0	30. jun. 2008
programmer 	hugo
tested by	oscat

FT_PI is a PI controller with manual functionality.
The PID controller works according to the fomula Y = e *(KP+ KI * INTEG(e) ) + offset, while e = set_point - actual.
a rst will reset all internal data, while a switch to manual will cause the controller to follow the function Y = manual_in + offset.
limit_h and Limit_l set the possible output range of Y.
the output flags lim will signal that the output limits are active.

*)

(* @END_DECLARATION := '0' *)
DIFF := CTRL_IN(SET0, ACT, SUP);
pid(in := DIFF, kp := KP, tn := TN, tv := TV, lim_l := LL, lim_h := LH, rst := RST);
co(ci := pid.Y, OFFSET := OFS, man_in := M_I, lim_l := LL, lim_h := LH, MANUAL := MAN);
Y := co.Y;
LIM := co.LIM;

(* revision history

hm 1.12.2006	 	rev 1.1
	changed algorithm to trapezregel for higher accuracy.

hm 3.1.2007		rev 1.2
	added integ_band to select when the integrator is active.

hm	3.3.2007		rev 1.3
	added default values to inputs KP, TN, TV, LIMIT_L und LIMIT_H.

hm 31.oct 2007	rev 1.4
	total rewrite of the module to avoid failures when one of the limits is 0

hm	3.11.2007	rev 1.5
	added noise input to filter noise
	added output diff
	set limit output false when output is within limits
	overfolw was not set correctly

hm	5. jan 2008	rev 1.6
	improved code for better performance
*)
END_FUNCTION_BLOCK

(* @NESTEDCOMMENTS := 'Yes' *)
(* @PATH := '\/Engineering\/control' *)
(* @OBJECTFLAGS := '0, 8' *)
(* @SYMFILEFLAGS := '2048' *)
FUNCTION_BLOCK CTRL_PWM
VAR_INPUT
	CI, MAN_IN : REAL;
	MANUAL : BOOL;
	F : REAL;
END_VAR
VAR_OUTPUT
	Q : BOOL;
END_VAR
VAR
	PW : PWM_DC;
END_VAR

(*
version 1.1	21. oct. 2008
programmer 	hugo
tested by	oscat

*)

(* @END_DECLARATION := '0' *)
PW(F := F, DC := SEL(MANUAL,CI,MAN_IN));
Q := PW.Q;

(* revision history
hm 3. jun. 2008 	rev 1.0
	original version

hm	21. oct. 2008	rev 1.1
	optimized code

*)
END_FUNCTION_BLOCK

(* @NESTEDCOMMENTS := 'Yes' *)
(* @PATH := '\/Engineering\/control' *)
(* @OBJECTFLAGS := '0, 8' *)
(* @SYMFILEFLAGS := '2048' *)
FUNCTION DEAD_BAND : REAL
VAR_INPUT
	X : REAL;
	L : REAL;
END_VAR

(*
version 1.2	18. jan. 2011
programmer 	hugo
tested by		oscat

DEAD_BAND ist eine lineare �bertragungsfunktion mit Totzone. Die Funktion verschiebt den positiven Teil der Kurve um +L und den negativen Teil der Kurve um -L.
DEAD_BAND = X - L wenn X > L)
DEAD_BAND = X + L wenn X < -L
DEAD_BAND = 0 wenn Abs(X) <= L

*)
(* @END_DECLARATION := '0' *)
IF X > L THEN
	DEAD_BAND := X - L;
ELSIF X < -L THEN
	DEAD_BAND := X + L;
ELSE
	DEAD_BAND := 0.0;
END_IF;

(* revision history
hm	2. nov. 2007	rev 1.0
	original version

hm	14. jun. 2008	rev 1.1
	improved performance

hm	18. jan. 2011	rev 1.2
	assign 0 before return
*)
END_FUNCTION

(* @NESTEDCOMMENTS := 'Yes' *)
(* @PATH := '\/Engineering\/control' *)
(* @OBJECTFLAGS := '0, 8' *)
(* @SYMFILEFLAGS := '2048' *)
FUNCTION_BLOCK DEAD_BAND_A
VAR_INPUT
	X : REAL;
	T : TIME;
	KL : REAL := 1.0;
	LM : REAL;
END_VAR
VAR_OUTPUT
	Y : REAL;
	L : REAL;
END_VAR
VAR
	tp1 : FT_PT1;
	tp2 : FT_PT1;
END_VAR

(*
version 1.1	11. mar. 2009
programmer 	hugo
tested by		oscat

DEAD_BAND ist eine lineare �bertragungsfunktion mit Totzone. Die Funktion verschiebt den positiven Teil der Kurve um -L und den negativen Teil der Kurve um +L.
DEAD_BAND = X wenn Abs(X) > L wenn Abs(X) > L
DEAD_BAND = 0 wenn Abs(X) <= L
Die Breite der Totzone wird automatisch aus dem Signalrauschen errechnet.

*)
(* @END_DECLARATION := '0' *)
(* filter the input signal *)
tp1(in := X, T:= T);

(* filter the HF portion to generate a stable L *)
tp2(in := ABS(tp1.out - X), T := MULTIME(T, 4.0));

(* now we determine L which is half the width of the dead band *)
L := MIN(KL * tp2.out, LM);

IF X > L THEN
	Y := X - L;
ELSIF X < -L THEN
	Y := X + L;
ELSE
	Y := 0.0;
END_IF;

(* revision history
hm	14. jun. 2008	rev 1.0
	original version

hm	11. mar. 2009	rev 1.1
	real constants updated to new systax using dot

*)
END_FUNCTION_BLOCK

(* @NESTEDCOMMENTS := 'Yes' *)
(* @PATH := '\/Engineering\/control' *)
(* @OBJECTFLAGS := '0, 8' *)
(* @SYMFILEFLAGS := '2048' *)
FUNCTION DEAD_ZONE : REAL
VAR_INPUT
	X : REAL;
	L : REAL;
END_VAR

(*
version 1.2	11. mar. 2009
programmer 	hugo
tested by		oscat

dead_zone2 is a linear transfer function which follows a linear function except for x is close to 0.
Y = X if abs(x) > L otherwise its 0.

*)
(* @END_DECLARATION := '0' *)
IF ABS(x) > L THEN
	dead_zone := X;
ELSE
	DEAD_ZONE := 0.0;
END_IF;

(* revision history
hm	12. feb. 2007	rev 1.0
	original version

hm	14. jun. 2008	rev 1.1
	improved performance

hm	11. mar. 2009	rev 1.2
	real constants updated to new systax using dot

*)
END_FUNCTION

(* @NESTEDCOMMENTS := 'Yes' *)
(* @PATH := '\/Engineering\/control' *)
(* @OBJECTFLAGS := '0, 8' *)
(* @SYMFILEFLAGS := '2048' *)
FUNCTION_BLOCK DEAD_ZONE2
VAR_INPUT
	X : REAL;
	L : REAL;
END_VAR
VAR_OUTPUT
	Y: REAL;
END_VAR

(*
version 1.1	11. mar. 2009
programmer 	hugo
tested by		tobias

dead_zone2 is a linear transfer function which follows a linear function except for x is close to 0.
Y = X if abs(x) > L.
for values of 0 +/- L a hysteresis function will hold the output at + or - L.

*)
(* @END_DECLARATION := '0' *)
IF ABS(x) > L THEN
	Y := X;
ELSIF Y > 0.0 THEN
	Y := L;
ELSE
	Y := -L;
END_IF;

(* revision history

hm	12. feb. 2007	rev 1.0
	original version

hm	11. mar. 2009	rev 1.1
	real constants updated to new systax using dot

*)

END_FUNCTION_BLOCK

(* @NESTEDCOMMENTS := 'Yes' *)
(* @PATH := '\/Engineering\/control' *)
(* @OBJECTFLAGS := '0, 8' *)
(* @SYMFILEFLAGS := '2048' *)
FUNCTION_BLOCK FT_DERIV
VAR_INPUT
	in : REAL;
	K : REAL := 1.0;
	run : BOOL := TRUE;
END_VAR
VAR_OUTPUT
	out : REAL;
END_VAR
VAR
	old: REAL;
	tx: DWORD;
	last: DWORD;
	init: BOOL;
	tc: REAL;
END_VAR

(*
version 1.5	11. mar. 2009
programmer 	hugo
tested by		oscat

FT_deriv calculates the derivate over the signal "in" with Faktor "K".
a run input enables or stops the calculation, if left unconnected its true and therfore the calculation is executed.
if K is not specified the default is 1.

*)

(* @END_DECLARATION := '0' *)
(* read system time *)
tx := T_PLC_US();
tc := DWORD_TO_REAL(tx - last);
last := tx;

(* init on first startup *)
IF NOT init THEN
	init := TRUE;
	old := in;
ELSIF run AND tc > 0.0 THEN
	out := (in - old) / tc * 1000000.0 * K;
	old := in;
ELSE
	out := 0.0;
END_IF;

(*
hm 3.1.2007			rev 1.1
	added init code for startup
	set the default for K to 1

hm	15. sep 2007	rev 1.2
	replaced Time() with T_PLC_US for compatibility and performance reasons
	increased accuracy and work in microseconds internally

hm 29 oct 2007	rev 1.3
	prohibit calculation when tx - last = 0 to avoid division by 0 and increase accuracy on fast systems

hm	6. nov. 2008	rev 1.4
	improved performance

hm	11. mar. 2009	rev 1.5
	inproved code
*)
END_FUNCTION_BLOCK

(* @NESTEDCOMMENTS := 'Yes' *)
(* @PATH := '\/Engineering\/control' *)
(* @OBJECTFLAGS := '0, 8' *)
(* @SYMFILEFLAGS := '2048' *)
FUNCTION_BLOCK FT_IMP
VAR_INPUT
	in : REAL;
	T : TIME;
	K : REAL := 1.0;
END_VAR
VAR_OUTPUT
	out : REAL;
END_VAR
VAR
	t1 : FT_PT1;
END_VAR

(*
version 1.1	3 Jan 2007
programmer 	hugo
tested by	oscat

FT_IMP is 	an impulse filter (high pass filter) with the time T and factor K.

*)
(* @END_DECLARATION := '0' *)
T1(in:= in, T:=T);
out := (in - t1.out) * K;

(*
hm 3.1.2007	rev 1.1
	added factor K

*)
END_FUNCTION_BLOCK

(* @NESTEDCOMMENTS := 'Yes' *)
(* @PATH := '\/Engineering\/control' *)
(* @OBJECTFLAGS := '0, 8' *)
(* @SYMFILEFLAGS := '2048' *)
FUNCTION_BLOCK FT_INT
VAR_INPUT
	IN : REAL;
	K : REAL := 1;
	RUN : BOOL := TRUE;
	RST : BOOL;
	OUT_MIN : REAL := -1E37;
	OUT_MAX : REAL := 1E37;
END_VAR
VAR_OUTPUT
	OUT : REAL;
	LIM : BOOL;
END_VAR
VAR
	INTeg : INTEGRATE;
END_VAR

(*
version 2.2	10. mar. 2009
programmer 	hugo
tested by		oscat

FT_int is an integrator with input IN and factor K.
integration is only done while run = true, if run is false integration is stopped and the out remains at the last value.
if run is left unconnected, run is considered true by the function block.
the output ET will display the total integration time from last reset.
the out_min and out_max values can be set to ,imit the output value range.
the default for K is 1.

*)
(* @END_DECLARATION := '0' *)
IF rst THEN
	out := 0.0;
ELSE
	integ(X := IN, E := RUN, K := K, Y := out);
END_IF;

(* limit the outputs *)
IF out >= OUT_MAX THEN
	out := out_max;
	LIM := TRUE;
ELSIF out <= out_min THEN
	out := out_min;
	lim := TRUE;
ELSE
	lim := FALSE;
END_IF;

(*
hm 13.12.2006	rev 1.1
	changed to "trapezregel" which increases accuracy
	before out := out + in * time new: out := out + (in + in_last) / 2 * time

hm 15.1.2007		rev 1.2
	added default for k to be 1.

hm	15.9.2007		rev 1.3
	replaced time() with T_PLC_US for compatibility and performance reason
	increased internal accuracy to microseconds

hm 29. oct 2007		rev 1.4
	changed code so int will not be called is time difference is 0 to increase accuracy on systems
	with cycle times below 1ms

hm	2. dec 2007	 	rev 1.5
	changed code for better performance

hm	5. jan 2008		rev 1.6
	further improvements in performance

hm	8. feb 2008		rev 1.7
	deleted limits +/- 1000 now limit is the range of real
	added variables out1 and out2 to extend the resolution
	corrected an error with elapsed time
	deleted unusfull output ET

hm	13. mar 2008	rev 1.8
	changed preset value out_min to -1e37.
	stop integrator at the limits.

hm	16. mar 2008	rev 1.9
	added type conversion to avoid warning under codesys 3.0

hm	2. jun. 2008	rev 2.0
	rewritten with clear code
	limits can now be set without run

hm	3. nov. 2008	rev 2.1
	optimized code using INTEGRATE and LIMX

hm	10. mar. 2009	rev 2.2
	removed nested comments
*)

END_FUNCTION_BLOCK

(* @NESTEDCOMMENTS := 'Yes' *)
(* @PATH := '\/Engineering\/control' *)
(* @OBJECTFLAGS := '0, 8' *)
(* @SYMFILEFLAGS := '2048' *)
FUNCTION_BLOCK FT_INT2
VAR_INPUT
	IN : REAL;
	K : REAL := 1.0;
	RUN : BOOL := TRUE;
	RST : BOOL;
	OUT_MIN : REAL := -1.0E38;
	OUT_MAX : REAL := 1.0E38;
END_VAR
VAR_OUTPUT
	OUT : REAL;
	LIM : BOOL;
END_VAR
VAR
	integ: INTEGRATE;
	ix : REAL;
	val : REAL2;
END_VAR

(*
version 1.2	11. mar. 2009
programmer 	hugo
tested by		oscat

FT_int2 is an integrator with input IN and factor K.
integration is only done while run = true, if run is false integration is stopped and the out remains at the last value.
if run is left unconnected, run is considered true by the function block.
the out_min and out_max values can be set to ,imit the output value range.
the default for K is 1.
FT_INT2 has double presision accuracy (14 digits).

*)
(* @END_DECLARATION := '0' *)
IF RST THEN
	val := R2_SET(0.0);
	out := 0.0;
ELSE
	integ(X := IN, E := RUN, K := K, Y := ix);
	val := R2_ADD(val, ix);
	ix := 0.0;
	OUT := val.RX;
END_IF;

(* check output for limits *)
IF out > OUT_MIN AND out < OUT_MAX THEN
	LIM := FALSE;
ELSE
	OUT := LIMIT(OUT_MIN, OUT, OUT_MAX);
	val := R2_SET(OUT);
	LIM := TRUE;
END_IF;

(*	revision history
hm	2. jun. 2008	rev 1.0
	original version

hm	5. nov. 2008	rev 1.1
	rewritten code using integrate

hm	11. mar. 2009	rev 1.2
	real constants updated to new systax using dot

*)

END_FUNCTION_BLOCK

(* @NESTEDCOMMENTS := 'Yes' *)
(* @PATH := '\/Engineering\/control' *)
(* @OBJECTFLAGS := '0, 8' *)
(* @SYMFILEFLAGS := '2048' *)
FUNCTION_BLOCK FT_PD
VAR_INPUT
	IN : REAL;
	KP : REAL := 1.0;
	TV : REAL := 1.0;
END_VAR
VAR_OUTPUT
	Y : REAL;
END_VAR
VAR
	diff : FT_DERIV;
END_VAR

(*
version 1.0	3. jun 2008
programmer 	hugo
tested by		tobias

FT_PD is a PD controller.
The PD controller works according to the fomula Y = KP *(IN + DERIV(e) ).

*)

(* @END_DECLARATION := '0' *)
(* run differentiator *)
diff(IN := IN, K := TV);

(* combine both values *)
Y := KP * (diff.out + IN);

(* revision history
hm 	3. jun. 2008 	rev 1.0
	original version

*)
END_FUNCTION_BLOCK

(* @NESTEDCOMMENTS := 'Yes' *)
(* @PATH := '\/Engineering\/control' *)
(* @OBJECTFLAGS := '0, 8' *)
(* @SYMFILEFLAGS := '2048' *)
FUNCTION_BLOCK FT_PDT1
VAR_INPUT
	IN : REAL;
	KP : REAL := 1.0;
	TV : REAL := 1.0;
	T1 : REAL := 1.0;
END_VAR
VAR_OUTPUT
	Y : REAL;
END_VAR
VAR
	diff : FT_DERIV;
	TP : FT_PT1;
END_VAR

(*
version 1.0	3. jun 2008
programmer 	hugo
tested by		tobias

FT_PD is a PD controller.
The PD controller works according to the fomula Y = KP *(IN + DERIV(e) ).

*)

(* @END_DECLARATION := '0' *)
(* run differentiator *)
diff(IN := IN, K := TV);

(* Run PT1 filter *)
tp(in := diff.out, T := REAL_TO_TIME(T1));

(* combine both values *)
Y := KP * (tp.out + IN);

(* revision history
hm 	3. jun. 2008 	rev 1.0
	original version

*)
END_FUNCTION_BLOCK

(* @NESTEDCOMMENTS := 'Yes' *)
(* @PATH := '\/Engineering\/control' *)
(* @OBJECTFLAGS := '0, 8' *)
(* @SYMFILEFLAGS := '2048' *)
FUNCTION_BLOCK FT_PI
VAR_INPUT
	IN : REAL;
	KP : REAL := 1.0;
	KI : REAL := 1.0;
	ILIM_L : REAL := -1E38;
	ILIM_H : REAL := 1E38;
	IEN : BOOL := TRUE;
	RST : BOOL;
END_VAR
VAR_OUTPUT
	Y : REAL;
	LIM : BOOL;
END_VAR
VAR
	integ : FT_INT;
END_VAR

(*
version 2.0	3. jun 2008
programmer 	hugo
tested by		tobias

FT_PI is a PI controller.
The PID controller works according to the fomula Y = IN *(KP+ KI * INTEG(e) ).
a rst will reset the integrator to 0
ilim_h and iLim_l set the possible output range of the internal integrator.
the output flags lim will signal that the output limits are active.

default values for KP = 1, KI = 1, ILIM_L = -1E37, iLIM_H = +1E38.
*)

(* @END_DECLARATION := '0' *)
(* run integrator *)
integ(IN := IN, K := KI, RUN := IEN, RST := RST, OUT_MIN := ILIM_L, OUT_MAX := ILIM_H);

(* check if integrator has reached its limits and set overflow *)
LIM := integ.LIM;
Y := KP * IN + integ.Out;

(* revision history
hm 	3. jun. 2008 	rev 2.0
	original version

*)
END_FUNCTION_BLOCK

(* @NESTEDCOMMENTS := 'Yes' *)
(* @PATH := '\/Engineering\/control' *)
(* @OBJECTFLAGS := '0, 8' *)
(* @SYMFILEFLAGS := '2048' *)
FUNCTION_BLOCK FT_PID
VAR_INPUT
	IN : REAL;
	KP : REAL := 1.0;
	TN : REAL := 1.0;
	TV : REAL := 1.0;
	ILIM_L : REAL := -1.0E38;
	ILIM_H : REAL := 1.0E38;
	IEN : BOOL := TRUE;
	RST : BOOL;
END_VAR
VAR_OUTPUT
	Y : REAL;
	LIM : BOOL;
END_VAR
VAR
	integ : FT_INT;
	diff : FT_DERIV;
END_VAR

(*
version 2.1	11. mar. 2009
programmer 	hugo
tested by		tobias

FT_PI is a PI controller.
The PID controller works according to the fomula Y = IN *(KP+ KI * INTEG(e) ).
a rst will reset the integrator to 0
ilim_h and iLim_l set the possible output range of the internal integrator.
the output flags lim will signal that the output limits are active.

default values for KP = 1, KI = 1, ILIM_L = -1E37, iLIM_H = +1E38.
*)

(* @END_DECLARATION := '0' *)
(* run integrator only if TN > 0 *)
IF TN > 0.0 THEN
	integ(IN := IN, K := 1.0 / TN, RUN := IEN, RST := RST, OUT_MIN := ILIM_L, OUT_MAX := ILIM_H);
ELSE
	integ(RST := FALSE);
END_IF;

(* run differentiator *)
diff(IN := IN, K := TV);

(* combine both values *)
Y := KP * (integ.Out + diff.out + IN);

(* check if integrator has reached its limits and set overflow *)
LIM := integ.LIM;

(* revision history
hm 3. jun. 2008 	rev 2.0
	original version

hm	11. mar. 2009	rev 2.1
	real constants updated to new systax using dot

*)
END_FUNCTION_BLOCK

(* @NESTEDCOMMENTS := 'Yes' *)
(* @PATH := '\/Engineering\/control' *)
(* @OBJECTFLAGS := '0, 8' *)
(* @SYMFILEFLAGS := '2048' *)
FUNCTION_BLOCK FT_PIDW
VAR_INPUT
	IN : REAL;
	KP : REAL := 1.0;
	TN : REAL := 1.0;
	TV : REAL := 1.0;
	LIM_L : REAL := -1.0E38;
	LIM_H : REAL := 1.0E38;
	RST : BOOL;
END_VAR
VAR_OUTPUT
	Y : REAL;
	LIM : BOOL;
END_VAR
VAR
	integ : INTEGRATE;
	diff : FT_DERIV;
	YI: REAL;
END_VAR

(*
version 1.2	11. mar. 2009
programmer 	hugo
tested by		oscat

FT_PIDW is a PID controller with dynamic wind_up reset.
The PID controller works according to the fomula Y = KP *(IN + KI * INTEG(e) + DERIV(e) ).
a rst will reset the integrator to 0
lim_h and Lim_l set the possible output range of the internal integrator.
the output flags lim will signal that the output limits are active.

default values for KP = 1, KI = 1, ILIM_L = -1E37, iLIM_H = +1E38.
*)

(* @END_DECLARATION := '0' *)
(* run the integrator *)
IF tn = 0.0 OR rst THEN
	integ(E := FALSE, Y := YI);
	YI := 0.0;
ELSE
	integ(X := IN, K := 1.0 / TN, E := NOT LIM, Y := YI);
END_IF;

(* add up integrator and linear part *)
Y := KP * (IN + YI);

(* run differentiator *)
diff(IN := IN, K := TV);

(* set lim before differentiator is added to stop integrator if necessary *)
IF Y > LIM_L AND Y < LIM_H THEN
	LIM := FALSE;
ELSE
	LIM := TRUE;
END_IF;

(* add differential part and limit output Y *)

Y := LIMIT(LIM_L, Y + KP * diff.out, LIM_H);

(* revision history
hm 3. jun. 2008 	rev 1.0
	original version

hm	5. nov. 2008	rev 1.1
	changed code to use integrate

hm	11. mar. 2009	rev 1.2
	real constants updated to new systax using dot

*)
END_FUNCTION_BLOCK

(* @NESTEDCOMMENTS := 'Yes' *)
(* @PATH := '\/Engineering\/control' *)
(* @OBJECTFLAGS := '0, 8' *)
(* @SYMFILEFLAGS := '2048' *)
FUNCTION_BLOCK FT_PIDWL
VAR_INPUT
	IN : REAL;
	KP : REAL := 1.0;
	TN : REAL := 1.0;
	TV : REAL := 1.0;
	LIM_L : REAL := -1.0E38;
	LIM_H : REAL := 1.0E38;
	RST : BOOL;
END_VAR
VAR_OUTPUT
	Y : REAL;
	LIM : BOOL;
END_VAR
VAR
	piwl : FT_PIWL;
	diff : FT_DERIV;
END_VAR

(*
version 1.3	13. nov. 2009
programmer 	hugo
tested by		tobias

FT_PIDWL is a PID controller with dynamic wind_up reset.
The PID controller works according to the fomula Y = KP *(IN + KI * INTEG(e) + DERIV(e) ).
a rst will reset the integrator to 0
lim_h and Lim_l set the possible output range of the internal integrator.
the output flags lim will signal that the output limits are active.

default values for KP = 1, KI = 1, ILIM_L = -1E37, iLIM_H = +1E38.
*)

(* @END_DECLARATION := '0' *)
(* if rst then *)
IF rst THEN
	piwl(rst := TRUE);
	piwl.RST := FALSE;
ELSE
	(* run PIWL controller first *)
	(* we need to check if TN = 0 and do alternative calls *)
	IF TN = 0.0 THEN
		piwl(in := IN * KP, KP := 1.0, KI := 0.0, LIM_L := LIM_L, LIM_H := LIM_H);
	ELSE
		piwl(in := IN * KP, KP := 1.0, KI := 1.0 / TN, LIM_L := LIM_L, LIM_H := LIM_H);
	END_IF;

	(* run differentiator and add_to_output *)
	diff(IN := IN, K := KP * TV);
	Y := piwl.Y + diff.out;

	(* limit the output *)
	IF Y < LIM_L THEN
		LIM := TRUE;
		Y := LIM_L;
	ELSIF Y > LIM_H THEN
		LIM := TRUE;
		Y := LIM_H;
	ELSE
		LIM := FALSE;
	END_IF;
END_IF;

(* revision history
hm 13. jun. 2008 	rev 1.0
	original version

hm	25. jan 2008	rev 1.1
	multiply differential part with KP

hm	11. mar. 2009	rev 1.2
	real constants updated to new systax using dot

hm	13. nov. 2009	rev 1.3
	fixed code for negative KP

*)
END_FUNCTION_BLOCK

(* @NESTEDCOMMENTS := 'Yes' *)
(* @PATH := '\/Engineering\/control' *)
(* @OBJECTFLAGS := '0, 8' *)
(* @SYMFILEFLAGS := '2048' *)
FUNCTION_BLOCK FT_PIW
VAR_INPUT
	IN : REAL;
	KP : REAL := 1.0;
	KI : REAL := 1.0;
	LIM_L : REAL := -1E38;
	LIM_H : REAL := 1E38;
	RST : BOOL;
END_VAR
VAR_OUTPUT
	Y : REAL;
	LIM : BOOL;
END_VAR
VAR
	integ : FT_INT;
END_VAR

(*
version 1.0	3. jun 2008
programmer 	hugo
tested by		tobias

FT_PIW is a PI controller.
The PID controller works according to the fomula Y = IN *(KP+ KI * INTEG(e) ).
a rst will reset the integrator to 0
ilim_h and iLim_l set the possible output range of the internal integrator.
the output flag lim will signal that the output limits are active.
the controller is equipped with anti wind_up circuitry that stops the integrator when lim_h or lim_l is reached

default values for KP = 1, KI = 1, ILIM_L = -1E37, iLIM_H = +1E38.
*)

(* @END_DECLARATION := '0' *)
(* run integrator *)
integ(IN := IN, K := KI, RUN := NOT LIM, RST := RST);

(* set output value *)
Y := KP * IN + integ.Out;

(* check for limits and set integrator for anti wind up *)
IF Y < LIM_L THEN
	Y := LIM_L;
	LIM := TRUE;
ELSIF Y > LIM_H THEN
	Y := LIM_H;
	LIM := TRUE;
ELSE
	LIM := FALSE;
END_IF;

(* revision history
hm 	3. jun. 2008 	rev 1.0
	original version

*)
END_FUNCTION_BLOCK

(* @NESTEDCOMMENTS := 'Yes' *)
(* @PATH := '\/Engineering\/control' *)
(* @OBJECTFLAGS := '0, 8' *)
(* @SYMFILEFLAGS := '2048' *)
FUNCTION_BLOCK FT_PIWL
VAR_INPUT
	IN : REAL;
	KP : REAL := 1.0;
	KI : REAL := 1.0;
	LIM_L : REAL := -1.0E38;
	LIM_H : REAL := 1.0E38;
	RST : BOOL;
END_VAR
VAR_OUTPUT
	Y : REAL;
	LIM : BOOL;
END_VAR
VAR
	init: BOOL;
	tx: DWORD;
	tc : REAL;
	t_last: DWORD;
	in_last : REAL;
	i: REAL;
	p: REAL;
END_VAR

(*
version 1.3	11. mar. 2009
programmer 	hugo
tested by		oscat

FT_PIWL is a PI controller.
The PID controller works according to the fomula Y = IN *(KP+ KI * INTEG(e) ).
a rst will reset the integrator to 0
lim_h and Lim_l set the possible output range of the controller.
the output flag lim will signal that the output limits are active.
the integrator ist equipped with anti wind-up circuitry which limits trhe total output ranke to lim_l and lim_h

default values for KP = 1, KI = 1, ILIM_L = -1E37, iLIM_H = +1E38.
*)

(* @END_DECLARATION := '0' *)
(* initialize at power_up *)
IF NOT init OR RST THEN
	init := TRUE;
	in_last := in;
	t_last := T_PLC_US();
	i := 0.0;
	tc := 0.0;
ELSE
	(* read last cycle time in Microseconds *)
	tx := T_PLC_US();
	tc := DWORD_TO_REAL(tx - t_last);
	t_last := tx;

	(* calculate proportional part *)
	p := KP * IN;

	(* run integrator *)
	i := (IN + in_last) * 5.0E-7 * KI * tc + i;
	in_last := IN;

	(* calculate output Y *)
	Y := p + i;

	(* check output for limits *)
	IF Y >= LIM_H THEN
		Y := LIM_H;
		IF ki <> 0.0 THEN
			i := LIM_H - p;
		ELSE
			i := 0.0;
		END_IF;
		LIM := TRUE;
	ELSIF Y <= LIM_L THEN
		Y := LIM_L;
		IF ki <> 0.0 THEN
			i := LIM_L - p;
		ELSE
			i := 0.0;
		END_IF;
		LIM := TRUE;
	ELSE
		LIM := FALSE;
	END_IF;
END_IF;

(* revision history
hm 13. jun. 2008 	rev 1.0
	original version

hm	27. oct. 2008	rev 1.1
	integrator will not be adjusted when ki = 0

hm	25. jan 2009	rev 1.2
	module will also work with negative K

hm	11. mar. 2009	rev 1.3
	real constants updated to new systax using dot

*)
END_FUNCTION_BLOCK

(* @NESTEDCOMMENTS := 'Yes' *)
(* @PATH := '\/Engineering\/control' *)
(* @OBJECTFLAGS := '0, 8' *)
(* @SYMFILEFLAGS := '2048' *)
FUNCTION_BLOCK FT_PT1
VAR_INPUT
	in : REAL;
	T : TIME;
	K : REAL := 1.0;
END_VAR
VAR_OUTPUT
	out : REAL;
END_VAR
VAR
	last : DWORD;
	tx: DWORD;
	init: BOOL;
END_VAR

(*
version 1.11	18. jan. 2011
programmer 	hugo
tested by		oscat

FT_PT1 is an low pass filter with a programmable time T and faktor K.

*)
(* @END_DECLARATION := '0' *)
(* read system time *)
tx := T_PLC_US();

(* startup initialisation *)
IF NOT init OR T = t#0s THEN
	init := TRUE;
	out := K * in;
ELSE
	out := out + (in * K - out) * DWORD_TO_REAL(Tx - last) / TIME_TO_REAL(T) * 1.0E-3;
	IF ABS(out) < 1.0E-20 THEN out := 0.0; END_IF;
END_IF;
last := tx;

(*
hm 1.1.2007	rev 1.1
	corrected error while startup value was not correct
	for very small time values real output would run out of range.

hm 3.1.2007	rev 1.2
	corrected an error for falling edge failures.
	added output faktor K.

hm 27. 2. 2007	rev 1.3
	output will be input during init for definitive startup condition.

hm	15.9.2007	rev 1.4
	changed time() to T_PLC_US() for compatibilitxy resons
	increased internal accuracy to Microseconds instead of Milliseconds

hm	23. oct 2007	rev 1.5
	added out := in to the init statements

hm	30. nov 2007	rev 1.6
	changed out to be K * in during initialization

hm	5. jan 2008	rev 1.7
	improved code for better performance

hm	16. mar. 2008	rev 1.8
	added type conversion to avoid warning under codesys 3.0

hm	14. jun. 2008	rev 1.9
	improved code

hm	11. mar. 2009	rev 1.10
	real constants updated to new systax using dot

hm	18. jan. 2011	rev 1.11
	avoid underrun of out
*)
END_FUNCTION_BLOCK

(* @NESTEDCOMMENTS := 'Yes' *)
(* @PATH := '\/Engineering\/control' *)
(* @OBJECTFLAGS := '0, 8' *)
(* @SYMFILEFLAGS := '2048' *)
FUNCTION_BLOCK FT_PT2
VAR_INPUT
	in : REAL;
	T : TIME;
	D : REAL;
	K : REAL := 1.0;
END_VAR
VAR_OUTPUT
	out : REAL;
END_VAR
VAR
	init: BOOL;
	int1 : INTEGRATE;
	int2 : INTEGRATE;
	tn: REAL;
	I1, I2 : REAL;
	tn2: REAL;
END_VAR

(*
version 1.5	11. mar. 2009
programmer 	hugo
tested by		oscat

FT_PT2 is a 2nd grade filter with programmable times T, D and faktor K.

*)
(* @END_DECLARATION := '0' *)
(* startup initialisation *)
IF NOT init OR T = T#0s THEN
	init := TRUE;
	out := K * in;
	I2 := out;
ELSE
	TN := TIME_TO_REAL(T) * 1.0E-3;
	tn2 := TN * TN;
	int1(X := in * K / tn2 - I1 * 0.5 * D / TN - I2 / TN2, Y := I1);
	int2(X := I1,Y := I2);
	out := I2;
END_IF;

(* revision history

15.1.2007 hm		rev 1.1
	changed formula to new more acurate formula

hm 15.9.2007		rev 1.2
	deleted unused code for init system time reading tx

hm	30.11.2007	rev 1.3
	changed out to be K * in during initialization
	avoind divide by 0 if tn = 0

hm	3. nov. 2008	rev 1.4
	optimized code and fixed a problem with init

hm	11. mar. 2009	rev 1.5
	real constants updated to new systax using dot

*)
END_FUNCTION_BLOCK

(* @NESTEDCOMMENTS := 'Yes' *)
(* @PATH := '\/Engineering\/control' *)
(* @OBJECTFLAGS := '0, 8' *)
(* @SYMFILEFLAGS := '2048' *)
FUNCTION_BLOCK FT_TN16
VAR_INPUT
	in : REAL;
	T : TIME;
END_VAR
VAR_OUTPUT
	out : REAL;
	trig : BOOL;
END_VAR
VAR
	length : INT := 16;
	X : ARRAY[0..15] OF REAL;
	cnt : INT;
	last : TIME;
	tx: TIME;
	init: BOOL;
END_VAR

(*
version 1.1	16 sep 2007
programmer 	hugo
tested by		tobias

FT_TN16 is delay function, it will delay a signal by a specified time : T and will store 16 values of in before they are put thru to out.
for higher or lower resolution please use FT_TN8 or FT_TN64 instead.

*)
(* @END_DECLARATION := '0' *)
(* read system time *)
tx := DWORD_TO_TIME(T_PLC_MS());

trig := FALSE;
IF NOT init THEN
	x[cnt] := in;
	init := TRUE;
	last := tx;
ELSIF tx - last >= T / length THEN
	IF cnt = length - 1 THEN cnt := 0; ELSE cnt := cnt + 1; END_IF;
	Out := X[cnt];
	x[cnt] := in;
	last := tx;
	Trig := TRUE;
END_IF;

(* revision history
hm		1. jan 2007	rev 1.0
	original version

hm		16. sep 2007	rev 1.1
	changes time() to T_plc_ms() for compatibility reasons

*)
END_FUNCTION_BLOCK

(* @NESTEDCOMMENTS := 'Yes' *)
(* @PATH := '\/Engineering\/control' *)
(* @OBJECTFLAGS := '0, 8' *)
(* @SYMFILEFLAGS := '2048' *)
FUNCTION_BLOCK FT_TN64
VAR_INPUT
	in : REAL;
	T : TIME;
END_VAR
VAR_OUTPUT
	out : REAL;
	trig: BOOL;
END_VAR
VAR
	length : INT := 64;
	X : ARRAY[0..63] OF REAL;
	cnt : INT;
	last : TIME;
	tx: TIME;
	init: BOOL;
END_VAR
